LIN {X 0,Y 409.441,Z 300.015,A -85,B 0,C 180,E1 20196.049,E2 20196.049} C_VEL
LIN {X 0,Y 414.724,Z 318.91,A -85,B 0,C 180,E1 20192.601,E2 20192.601} C_VEL
LIN {X 0,Y 418.391,Z 333.673,A -85,B 0,C 180,E1 20190.048,E2 20190.048} C_VEL
LIN {X 0,Y 416.064,Z 361.542,A -85,B 0,C 180,E1 20186.001,E2 20186.001} C_VEL
LIN {X 0,Y 414.003,Z 389.743,A -85,B 0,C 180,E1 20181.965,E2 20181.965} C_VEL
LIN {X 0,Y 413.216,Z 403.009,A -85,B 0,C 180,E1 20180.124,E2 20180.124} C_VEL
LIN {X 0,Y 416.515,Z 427.421,A -85,B 0,C 180,E1 20179.379,E2 20179.379} C_VEL
LIN {X 0,Y 413.998,Z 526.951,A -85,B 0,C 180,E1 20177.125,E2 20177.125} C_VEL
LIN {X 0,Y 413.552,Z 542.343,A -85,B 0,C 180,E1 20176.538,E2 20176.538} C_VEL
LIN {X 0,Y 412.934,Z 558.221,A -85,B 0,C 180,E1 20175.661,E2 20175.661} C_VEL
LIN {X 0,Y 412.172,Z 574.05,A -85,B 0,C 180,E1 20174.467,E2 20174.467} C_VEL
LIN {X 0,Y 411.427,Z 588.228,A -85,B 0,C 180,E1 20173.06,E2 20173.06} C_VEL
LIN {X 0,Y 410.741,Z 600.404,A -85,B 0,C 180,E1 20171.512,E2 20171.512} C_VEL
LIN {X 0,Y 410.206,Z 610.147,A -85,B 0,C 180,E1 20169.963,E2 20169.963} C_VEL
LIN {X 0,Y 409.748,Z 619.266,A -85,B 0,C 180,E1 20168.134,E2 20168.134} C_VEL
LIN {X 0,Y 409.435,Z 626.69,A -85,B 0,C 180,E1 20166.166,E2 20166.166} C_VEL
LIN {X 0,Y 409.281,Z 631.788,A -85,B 0,C 180,E1 20164.341,E2 20164.341} C_VEL
LIN {X 0,Y 409.227,Z 635.7,A -85,B 0,C 180,E1 20162.238,E2 20162.238} C_VEL
LIN {X 0,Y 409.285,Z 637.574,A -85,B 0,C 180,E1 20160.278,E2 20160.278} C_VEL
LIN {X 0,Y 409.451,Z 637.785,A -85,B 0,C 180,E1 20158.179,E2 20158.179} C_VEL
LIN {X 0,Y 409.729,Z 636.027,A -85,B 0,C 180,E1 20156.08,E2 20156.08} C_VEL
LIN {X 0,Y 410.14,Z 632.531,A -85,B 0,C 180,E1 20154.073,E2 20154.073} C_VEL
LIN {X 0,Y 410.724,Z 626.914,A -85,B 0,C 180,E1 20152.022,E2 20152.022} C_VEL
LIN {X 0,Y 411.417,Z 619.96,A -85,B 0,C 180,E1 20150.203,E2 20150.203} C_VEL
LIN {X 0,Y 412.286,Z 611.32,A -85,B 0,C 180,E1 20148.457,E2 20148.457} C_VEL
LIN {X 0,Y 413.331,Z 600.124,A -85,B 0,C 180,E1 20146.713,E2 20146.713} C_VEL
LIN {X 0,Y 414.344,Z 588.102,A -85,B 0,C 180,E1 20145.249,E2 20145.249} C_VEL
LIN {X 0,Y 415.388,Z 575.258,A -85,B 0,C 180,E1 20144,E2 20144} C_VEL
LIN {X 0,Y 416.433,Z 560.28,A -85,B 0,C 180,E1 20142.865,E2 20142.865} C_VEL
LIN {X 0,Y 417.393,Z 543.508,A -85,B 0,C 180,E1 20141.926,E2 20141.926} C_VEL
LIN {X 0,Y 418.191,Z 525.443,A -85,B 0,C 180,E1 20141.231,E2 20141.231} C_VEL
LIN {X 0,Y 424.218,Z 435.023,A -85,B 0,C 180,E1 20138.466,E2 20138.466} C_VEL
LIN {X 0,Y 424.373,Z 429.953,A -85,B 0,C 180,E1 20138.28,E2 20138.28} C_VEL
LIN {X 0,Y 421.463,Z 411.862,A -85,B 0,C 180,E1 20137.24,E2 20137.24} C_VEL
LIN {X 0,Y 419.727,Z 402.661,A -85,B 0,C 180,E1 20136.631,E2 20136.631} C_VEL
LIN {X 0,Y 423.555,Z 377.639,A -85,B 0,C 180,E1 20132.575,E2 20132.575} C_VEL
LIN {X 0,Y 428.286,Z 354.651,A -85,B 0,C 180,E1 20128.626,E2 20128.626} C_VEL
LIN {X 0,Y 429.025,Z 351.42,A -85,B 0,C 180,E1 20128.03,E2 20128.03} C_VEL
LIN {X 0,Y 427.636,Z 343.386,A -85,B 0,C 180,E1 20125.701,E2 20125.701} C_VEL
LIN {X 0,Y 426.273,Z 337.13,A -85,B 0,C 180,E1 20123.341,E2 20123.341} C_VEL
LIN {X 0,Y 425.312,Z 333.711,A -85,B 0,C 180,E1 20121.523,E2 20121.523} C_VEL
LIN {X 0,Y 424.901,Z 331.733,A -85,B 0,C 180,E1 20120.098,E2 20120.098} C_VEL
LIN {X 0,Y 424.618,Z 330.119,A -85,B 0,C 180,E1 20117.48,E2 20117.48} C_VEL
LIN {X 0,Y 424.896,Z 330.575,A -85,B 0,C 180,E1 20115.66,E2 20115.66} C_VEL
LIN {X 0,Y 426.204,Z 333.163,A -85,B 0,C 180,E1 20113.146,E2 20113.146} C_VEL
LIN {X 0,Y 427.711,Z 337.595,A -85,B 0,C 180,E1 20111.064,E2 20111.064} C_VEL
LIN {X 0,Y 429.535,Z 343.22,A -85,B 0,C 180,E1 20109.18,E2 20109.18} C_VEL
LIN {X 0,Y 431.487,Z 350.329,A -85,B 0,C 180,E1 20107.361,E2 20107.361} C_VEL
LIN {X 0,Y 432.028,Z 352.863,A -85,B 0,C 180,E1 20106.829,E2 20106.829} C_VEL
LIN {X 0,Y 426.646,Z 376.903,A -85,B 0,C 180,E1 20103.902,E2 20103.902} C_VEL
LIN {X 0,Y 424.049,Z 392.881,A -85,B 0,C 180,E1 20102.112,E2 20102.112} C_VEL
LIN {X 0,Y 425.783,Z 409.021,A -85,B 0,C 180,E1 20101.466,E2 20101.466} C_VEL
LIN {X 0,Y 425.816,Z 416.278,A -85,B 0,C 180,E1 20101.257,E2 20101.257} C_VEL
LIN {X 0,Y 421.996,Z 515.171,A -85,B 0,C 180,E1 20099.047,E2 20099.047} C_VEL
LIN {X 0,Y 419.948,Z 585.828,A -85,B 0,C 180,E1 20097.578,E2 20097.578} C_VEL
LIN {X 0,Y 418.736,Z 605.858,A -85,B 0,C 180,E1 20096.904,E2 20096.904} C_VEL
LIN {X 0,Y 417.429,Z 623.258,A -85,B 0,C 180,E1 20096.072,E2 20096.072} C_VEL
LIN {X 0,Y 415.921,Z 641.014,A -85,B 0,C 180,E1 20094.963,E2 20094.963} C_VEL
LIN {X 0,Y 414.353,Z 658.072,A -85,B 0,C 180,E1 20093.615,E2 20093.615} C_VEL
LIN {X 0,Y 412.829,Z 674.111,A -85,B 0,C 180,E1 20092.05,E2 20092.05} C_VEL
LIN {X 0,Y 411.475,Z 689.013,A -85,B 0,C 180,E1 20090.287,E2 20090.287} C_VEL
LIN {X 0,Y 410.322,Z 702.807,A -85,B 0,C 180,E1 20088.322,E2 20088.322} C_VEL
LIN {X 0,Y 409.422,Z 715.375,A -85,B 0,C 180,E1 20086.166,E2 20086.166} C_VEL
LIN {X 0,Y 408.847,Z 726.454,A -85,B 0,C 180,E1 20083.856,E2 20083.856} C_VEL
LIN {X 0,Y 408.556,Z 735.338,A -85,B 0,C 180,E1 20081.578,E2 20081.578} C_VEL
LIN {X 0,Y 408.504,Z 742.848,A -85,B 0,C 180,E1 20079.155,E2 20079.155} C_VEL
LIN {X 0,Y 408.585,Z 748.491,A -85,B 0,C 180,E1 20076.747,E2 20076.747} C_VEL
LIN {X 0,Y 408.725,Z 752.398,A -85,B 0,C 180,E1 20074.35,E2 20074.35} C_VEL
LIN {X 0,Y 408.841,Z 754.641,A -85,B 0,C 180,E1 20071.963,E2 20071.963} C_VEL
LIN {X 0,Y 408.862,Z 755.26,A -85,B 0,C 180,E1 20069.581,E2 20069.581} C_VEL
LIN {X 0,Y 408.779,Z 754.252,A -85,B 0,C 180,E1 20067.197,E2 20067.197} C_VEL
LIN {X 0,Y 408.628,Z 751.594,A -85,B 0,C 180,E1 20064.801,E2 20064.801} C_VEL
LIN {X 0,Y 408.496,Z 747.256,A -85,B 0,C 180,E1 20062.406,E2 20062.406} C_VEL
LIN {X 0,Y 408.465,Z 741.108,A -85,B 0,C 180,E1 20059.992,E2 20059.992} C_VEL
LIN {X 0,Y 408.614,Z 732.997,A -85,B 0,C 180,E1 20057.566,E2 20057.566} C_VEL
LIN {X 0,Y 409.04,Z 723.353,A -85,B 0,C 180,E1 20055.274,E2 20055.274} C_VEL
LIN {X 0,Y 409.742,Z 711.86,A -85,B 0,C 180,E1 20053.054,E2 20053.054} C_VEL
LIN {X 0,Y 410.71,Z 699.143,A -85,B 0,C 180,E1 20051.036,E2 20051.036} C_VEL
LIN {X 0,Y 411.906,Z 684.831,A -85,B 0,C 180,E1 20049.157,E2 20049.157} C_VEL
LIN {X 0,Y 413.227,Z 669.717,A -85,B 0,C 180,E1 20047.525,E2 20047.525} C_VEL
LIN {X 0,Y 414.612,Z 653.545,A -85,B 0,C 180,E1 20046.101,E2 20046.101} C_VEL
LIN {X 0,Y 415.964,Z 636.517,A -85,B 0,C 180,E1 20044.898,E2 20044.898} C_VEL
LIN {X 0,Y 417.227,Z 618.592,A -85,B 0,C 180,E1 20043.914,E2 20043.914} C_VEL
LIN {X 0,Y 418.356,Z 599.425,A -85,B 0,C 180,E1 20043.148,E2 20043.148} C_VEL
LIN {X 0,Y 419.065,Z 580.405,A -85,B 0,C 180,E1 20042.65,E2 20042.65} C_VEL
LIN {X 0,Y 422.694,Z 411.284,A -85,B 0,C 180,E1 20039.443,E2 20039.443} C_VEL
LIN {X 0,Y 420.158,Z 388.361,A -85,B 0,C 180,E1 20038.811,E2 20038.811} C_VEL
LIN {X 0,Y 424.415,Z 345.859,A -85,B 0,C 180,E1 20034.601,E2 20034.601} C_VEL
LIN {X 0,Y 424.551,Z 343.397,A -85,B 0,C 180,E1 20034.343,E2 20034.343} C_VEL
LIN {X 0,Y 416.406,Z 319.629,A -85,B 0,C 180,E1 20031.017,E2 20031.017} C_VEL
LIN {X 0,Y 409.402,Z 299.802,A -85,B 0,C 180,E1 20027.998,E2 20027.998} C_VEL
LIN {X 0,Y 409.391,Z 299.803,A -85,B 0,C 180,E1 20024.109,E2 20024.109} C_VEL
LIN {X 0,Y 409.376,Z 299.804,A -85,B 0,C 180,E1 20020.335,E2 20020.335} C_VEL
LIN {X 0,Y 409.367,Z 299.801,A -85,B 0,C 180,E1 20016.53,E2 20016.53} C_VEL
LIN {X 0,Y 409.368,Z 299.8,A -85,B 0,C 180,E1 20012.67,E2 20012.67} C_VEL
LIN {X 0,Y 409.371,Z 299.8,A -85,B 0,C 180,E1 20008.74,E2 20008.74} C_VEL
LIN {X 0,Y 409.373,Z 299.8,A -85,B 0,C 180,E1 20004.842,E2 20004.842} C_VEL
LIN {X 0,Y 409.381,Z 299.8,A -85,B 0,C 180,E1 20001.042,E2 20001.042} C_VEL
LIN {X 0,Y 409.398,Z 299.799,A -85,B 0,C 180,E1 19997.273,E2 19997.273} C_VEL
LIN {X 0,Y 409.423,Z 299.8,A -85,B 0,C 180,E1 19993.561,E2 19993.561} C_VEL
LIN {X 0,Y 409.42,Z 299.8,A -85,B 0,C 180,E1 19989.561,E2 19989.561} C_VEL
LIN {X 0,Y 409.416,Z 299.801,A -85,B 0,C 180,E1 19985.748,E2 19985.748} C_VEL
LIN {X 0,Y 409.411,Z 299.8,A -85,B 0,C 180,E1 19981.821,E2 19981.821} C_VEL
LIN {X 0,Y 409.393,Z 299.8,A -85,B 0,C 180,E1 19978.043,E2 19978.043} C_VEL
LIN {X 0,Y 409.382,Z 299.8,A -85,B 0,C 180,E1 19974.255,E2 19974.255} C_VEL
LIN {X 0,Y 409.379,Z 299.799,A -85,B 0,C 180,E1 19970.442,E2 19970.442} C_VEL
LIN {X 0,Y 409.381,Z 299.799,A -85,B 0,C 180,E1 19966.586,E2 19966.586} C_VEL
LIN {X 0,Y 409.386,Z 299.798,A -85,B 0,C 180,E1 19962.733,E2 19962.733} C_VEL
LIN {X 0,Y 409.393,Z 299.798,A -85,B 0,C 180,E1 19958.897,E2 19958.897} C_VEL
LIN {X 0,Y 409.414,Z 299.797,A -85,B 0,C 180,E1 19955.165,E2 19955.165} C_VEL
LIN {X 0,Y 409.424,Z 299.797,A -85,B 0,C 180,E1 19951.246,E2 19951.246} C_VEL
LIN {X 0,Y 409.431,Z 299.798,A -85,B 0,C 180,E1 19947.34,E2 19947.34} C_VEL
LIN {X 0,Y 409.43,Z 299.799,A -85,B 0,C 180,E1 19943.429,E2 19943.429} C_VEL
LIN {X 0,Y 409.437,Z 299.799,A -85,B 0,C 180,E1 19939.494,E2 19939.494} C_VEL
LIN {X 0,Y 409.428,Z 299.8,A -85,B 0,C 180,E1 19935.485,E2 19935.485} C_VEL
LIN {X 0,Y 409.423,Z 299.8,A -85,B 0,C 180,E1 19931.624,E2 19931.624} C_VEL
LIN {X 0,Y 409.401,Z 299.799,A -85,B 0,C 180,E1 19927.927,E2 19927.927} C_VEL
LIN {X 0,Y 409.395,Z 299.798,A -85,B 0,C 180,E1 19924.118,E2 19924.118} C_VEL
LIN {X 0,Y 409.394,Z 299.798,A -85,B 0,C 180,E1 19920.205,E2 19920.205} C_VEL
LIN {X 0,Y 409.394,Z 299.797,A -85,B 0,C 180,E1 19916.329,E2 19916.329} C_VEL
LIN {X 0,Y 409.395,Z 299.797,A -85,B 0,C 180,E1 19912.394,E2 19912.394} C_VEL
LIN {X 0,Y 409.398,Z 299.797,A -85,B 0,C 180,E1 19908.51,E2 19908.51} C_VEL
LIN {X 0,Y 409.406,Z 299.796,A -85,B 0,C 180,E1 19904.713,E2 19904.713} C_VEL
LIN {X 0,Y 409.426,Z 299.796,A -85,B 0,C 180,E1 19900.98,E2 19900.98} C_VEL
LIN {X 0,Y 409.445,Z 299.795,A -85,B 0,C 180,E1 19897.153,E2 19897.153} C_VEL
LIN {X 0,Y 409.436,Z 299.797,A -85,B 0,C 180,E1 19893.219,E2 19893.219} C_VEL
LIN {X 0,Y 409.445,Z 299.797,A -85,B 0,C 180,E1 19889.299,E2 19889.299} C_VEL
LIN {X 0,Y 409.432,Z 299.8,A -85,B 0,C 180,E1 19885.377,E2 19885.377} C_VEL
LIN {X 0,Y 409.428,Z 299.799,A -85,B 0,C 180,E1 19881.489,E2 19881.489} C_VEL
LIN {X 0,Y 409.412,Z 299.798,A -85,B 0,C 180,E1 19877.741,E2 19877.741} C_VEL
LIN {X 0,Y 408.478,Z 299.923,A -85,B 0,C 180,E1 19876.663,E2 19876.663} C_VEL
LIN {X 0,Y 403.736,Z 300.514,A -85,B 0,C 180,E1 19874.553,E2 19874.553} C_VEL
LIN {X 0,Y 401.598,Z 300.773,A -85,B 0,C 180,E1 19873.149,E2 19873.149} C_VEL
LIN {X 0,Y 401.49,Z 300.784,A -85,B 0,C 180,E1 19872.83,E2 19872.83} C_VEL
LIN {X 0,Y 401.505,Z 300.783,A -85,B 0,C 180,E1 19868.985,E2 19868.985} C_VEL
LIN {X 0,Y 401.503,Z 300.784,A -85,B 0,C 180,E1 19865.014,E2 19865.014} C_VEL
LIN {X 0,Y 401.511,Z 300.784,A -85,B 0,C 180,E1 19861.11,E2 19861.11} C_VEL
LIN {X 0,Y 401.505,Z 300.785,A -85,B 0,C 180,E1 19857.119,E2 19857.119} C_VEL
LIN {X 0,Y 401.505,Z 300.784,A -85,B 0,C 180,E1 19853.066,E2 19853.066} C_VEL
LIN {X 0,Y 401.509,Z 300.784,A -85,B 0,C 180,E1 19849.084,E2 19849.084} C_VEL
LIN {X 0,Y 401.5,Z 300.788,A -85,B 0,C 180,E1 19845.189,E2 19845.189} C_VEL
LIN {X 0,Y 401.505,Z 300.787,A -85,B 0,C 180,E1 19841.229,E2 19841.229} C_VEL
LIN {X 0,Y 401.491,Z 300.788,A -85,B 0,C 180,E1 19837.397,E2 19837.397} C_VEL
LIN {X 0,Y 401.503,Z 300.865,A -85,B 0,C 180,E1 19836.611,E2 19836.611} C_VEL
LIN {X 0,Y 406.949,Z 320.456,A -85,B 0,C 180,E1 19832.968,E2 19832.968} C_VEL
LIN {X 0,Y 410.79,Z 335.895,A -85,B 0,C 180,E1 19830.251,E2 19830.251} C_VEL
LIN {X 0,Y 408.357,Z 363.768,A -85,B 0,C 180,E1 19826.147,E2 19826.147} C_VEL
LIN {X 0,Y 406.149,Z 392.506,A -85,B 0,C 180,E1 19821.972,E2 19821.972} C_VEL
LIN {X 0,Y 405.523,Z 402.833,A -85,B 0,C 180,E1 19820.519,E2 19820.519} C_VEL
LIN {X 0,Y 408.911,Z 428.375,A -85,B 0,C 180,E1 19819.715,E2 19819.715} C_VEL
LIN {X 0,Y 406.252,Z 527.745,A -85,B 0,C 180,E1 19817.392,E2 19817.392} C_VEL
LIN {X 0,Y 405.756,Z 543.832,A -85,B 0,C 180,E1 19816.754,E2 19816.754} C_VEL
LIN {X 0,Y 405.144,Z 558.966,A -85,B 0,C 180,E1 19815.896,E2 19815.896} C_VEL
LIN {X 0,Y 404.354,Z 574.826,A -85,B 0,C 180,E1 19814.68,E2 19814.68} C_VEL
LIN {X 0,Y 403.579,Z 589.06,A -85,B 0,C 180,E1 19813.246,E2 19813.246} C_VEL
LIN {X 0,Y 402.841,Z 601.812,A -85,B 0,C 180,E1 19811.596,E2 19811.596} C_VEL
LIN {X 0,Y 402.245,Z 612.27,A -85,B 0,C 180,E1 19809.873,E2 19809.873} C_VEL
LIN {X 0,Y 401.822,Z 620.594,A -85,B 0,C 180,E1 19808.152,E2 19808.152} C_VEL
LIN {X 0,Y 401.507,Z 628.02,A -85,B 0,C 180,E1 19806.145,E2 19806.145} C_VEL
LIN {X 0,Y 401.345,Z 633.398,A -85,B 0,C 180,E1 19804.141,E2 19804.141} C_VEL
LIN {X 0,Y 401.31,Z 636.994,A -85,B 0,C 180,E1 19802.14,E2 19802.14} C_VEL
LIN {X 0,Y 401.387,Z 638.913,A -85,B 0,C 180,E1 19799.998,E2 19799.998} C_VEL
LIN {X 0,Y 401.58,Z 639.044,A -85,B 0,C 180,E1 19798,E2 19798} C_VEL
LIN {X 0,Y 401.9,Z 637.26,A -85,B 0,C 180,E1 19795.861,E2 19795.861} C_VEL
LIN {X 0,Y 402.347,Z 633.821,A -85,B 0,C 180,E1 19793.864,E2 19793.864} C_VEL
LIN {X 0,Y 402.968,Z 628.538,A -85,B 0,C 180,E1 19791.868,E2 19791.868} C_VEL
LIN {X 0,Y 403.732,Z 621.742,A -85,B 0,C 180,E1 19790.015,E2 19790.015} C_VEL
LIN {X 0,Y 404.704,Z 612.815,A -85,B 0,C 180,E1 19788.165,E2 19788.165} C_VEL
LIN {X 0,Y 405.895,Z 601.238,A -85,B 0,C 180,E1 19786.319,E2 19786.319} C_VEL
LIN {X 0,Y 407.068,Z 588.654,A -85,B 0,C 180,E1 19784.761,E2 19784.761} C_VEL
LIN {X 0,Y 408.191,Z 575.598,A -85,B 0,C 180,E1 19783.491,E2 19783.491} C_VEL
LIN {X 0,Y 409.297,Z 560.926,A -85,B 0,C 180,E1 19782.366,E2 19782.366} C_VEL
LIN {X 0,Y 410.316,Z 545.116,A -85,B 0,C 180,E1 19781.449,E2 19781.449} C_VEL
LIN {X 0,Y 411.2,Z 527.167,A -85,B 0,C 180,E1 19780.724,E2 19780.724} C_VEL
LIN {X 0,Y 418.014,Z 433.46,A -85,B 0,C 180,E1 19777.747,E2 19777.747} C_VEL
LIN {X 0,Y 416.157,Z 419.167,A -85,B 0,C 180,E1 19776.928,E2 19776.928} C_VEL
LIN {X 0,Y 413.134,Z 402.466,A -85,B 0,C 180,E1 19775.78,E2 19775.78} C_VEL
LIN {X 0,Y 417.403,Z 377.958,A -85,B 0,C 180,E1 19771.685,E2 19771.685} C_VEL
LIN {X 0,Y 422.437,Z 356.26,A -85,B 0,C 180,E1 19767.821,E2 19767.821} C_VEL
LIN {X 0,Y 422.44,Z 354.305,A -85,B 0,C 180,E1 19767.339,E2 19767.339} C_VEL
LIN {X 0,Y 421.315,Z 347.222,A -85,B 0,C 180,E1 19765.113,E2 19765.113} C_VEL
LIN {X 0,Y 420.202,Z 341.819,A -85,B 0,C 180,E1 19762.857,E2 19762.857} C_VEL
LIN {X 0,Y 419.509,Z 338.644,A -85,B 0,C 180,E1 19760.987,E2 19760.987} C_VEL
LIN {X 0,Y 419.266,Z 337.346,A -85,B 0,C 180,E1 19759.916,E2 19759.916} C_VEL
LIN {X 0,Y 419.215,Z 335.944,A -85,B 0,C 180,E1 19757.175,E2 19757.175} C_VEL
LIN {X 0,Y 419.561,Z 336.796,A -85,B 0,C 180,E1 19755.25,E2 19755.25} C_VEL
LIN {X 0,Y 420.818,Z 339.472,A -85,B 0,C 180,E1 19752.961,E2 19752.961} C_VEL
LIN {X 0,Y 422.108,Z 343.366,A -85,B 0,C 180,E1 19751.125,E2 19751.125} C_VEL
LIN {X 0,Y 424.055,Z 349.661,A -85,B 0,C 180,E1 19749.018,E2 19749.018} C_VEL
LIN {X 0,Y 425.699,Z 356.545,A -85,B 0,C 180,E1 19747.3,E2 19747.3} C_VEL
LIN {X 0,Y 419.973,Z 380.043,A -85,B 0,C 180,E1 19744.351,E2 19744.351} C_VEL
LIN {X 0,Y 417.641,Z 393.224,A -85,B 0,C 180,E1 19742.833,E2 19742.833} C_VEL
LIN {X 0,Y 419.323,Z 408.99,A -85,B 0,C 180,E1 19742.147,E2 19742.147} C_VEL
LIN {X 0,Y 419.446,Z 416.244,A -85,B 0,C 180,E1 19741.917,E2 19741.917} C_VEL
LIN {X 0,Y 415.269,Z 512.08,A -85,B 0,C 180,E1 19739.687,E2 19739.687} C_VEL
LIN {X 0,Y 412.858,Z 585.335,A -85,B 0,C 180,E1 19738.098,E2 19738.098} C_VEL
LIN {X 0,Y 411.556,Z 605.144,A -85,B 0,C 180,E1 19737.411,E2 19737.411} C_VEL
LIN {X 0,Y 410.073,Z 623.422,A -85,B 0,C 180,E1 19736.511,E2 19736.511} C_VEL
LIN {X 0,Y 408.439,Z 641.077,A -85,B 0,C 180,E1 19735.367,E2 19735.367} C_VEL
LIN {X 0,Y 406.694,Z 658.491,A -85,B 0,C 180,E1 19733.933,E2 19733.933} C_VEL
LIN {X 0,Y 405.084,Z 674.231,A -85,B 0,C 180,E1 19732.342,E2 19732.342} C_VEL
LIN {X 0,Y 403.544,Z 690.013,A -85,B 0,C 180,E1 19730.397,E2 19730.397} C_VEL
LIN {X 0,Y 402.352,Z 703.428,A -85,B 0,C 180,E1 19728.398,E2 19728.398} C_VEL
LIN {X 0,Y 401.428,Z 715.696,A -85,B 0,C 180,E1 19726.199,E2 19726.199} C_VEL
LIN {X 0,Y 400.845,Z 726.469,A -85,B 0,C 180,E1 19723.856,E2 19723.856} C_VEL
LIN {X 0,Y 400.55,Z 735.646,A -85,B 0,C 180,E1 19721.374,E2 19721.374} C_VEL
LIN {X 0,Y 400.534,Z 742.819,A -85,B 0,C 180,E1 19718.905,E2 19718.905} C_VEL
LIN {X 0,Y 400.642,Z 748.165,A -85,B 0,C 180,E1 19716.449,E2 19716.449} C_VEL
LIN {X 0,Y 400.807,Z 751.795,A -85,B 0,C 180,E1 19714.006,E2 19714.006} C_VEL
LIN {X 0,Y 400.926,Z 753.752,A -85,B 0,C 180,E1 19711.573,E2 19711.573} C_VEL
LIN {X 0,Y 400.944,Z 754.057,A -85,B 0,C 180,E1 19709.144,E2 19709.144} C_VEL
LIN {X 0,Y 400.827,Z 752.717,A -85,B 0,C 180,E1 19706.712,E2 19706.712} C_VEL
LIN {X 0,Y 400.663,Z 749.719,A -85,B 0,C 180,E1 19704.272,E2 19704.272} C_VEL
LIN {X 0,Y 400.525,Z 744.996,A -85,B 0,C 180,E1 19701.821,E2 19701.821} C_VEL
LIN {X 0,Y 400.507,Z 738.437,A -85,B 0,C 180,E1 19699.355,E2 19699.355} C_VEL
LIN {X 0,Y 400.707,Z 730.421,A -85,B 0,C 180,E1 19697.024,E2 19697.024} C_VEL
LIN {X 0,Y 401.187,Z 720.393,A -85,B 0,C 180,E1 19694.683,E2 19694.683} C_VEL
LIN {X 0,Y 401.965,Z 708.826,A -85,B 0,C 180,E1 19692.485,E2 19692.485} C_VEL
LIN {X 0,Y 403.035,Z 695.667,A -85,B 0,C 180,E1 19690.434,E2 19690.434} C_VEL
LIN {X 0,Y 404.277,Z 681.457,A -85,B 0,C 180,E1 19688.606,E2 19688.606} C_VEL
LIN {X 0,Y 405.711,Z 665.612,A -85,B 0,C 180,E1 19686.932,E2 19686.932} C_VEL
LIN {X 0,Y 407.2,Z 648.692,A -85,B 0,C 180,E1 19685.484,E2 19685.484} C_VEL
LIN {X 0,Y 408.576,Z 631.813,A -85,B 0,C 180,E1 19684.334,E2 19684.334} C_VEL
LIN {X 0,Y 409.867,Z 613.454,A -85,B 0,C 180,E1 19683.37,E2 19683.37} C_VEL
LIN {X 0,Y 410.95,Z 594.557,A -85,B 0,C 180,E1 19682.663,E2 19682.663} C_VEL
LIN {X 0,Y 411.592,Z 574.104,A -85,B 0,C 180,E1 19682.184,E2 19682.184} C_VEL
LIN {X 0,Y 415.286,Z 412.136,A -85,B 0,C 180,E1 19679.039,E2 19679.039} C_VEL
LIN {X 0,Y 412.724,Z 388.405,A -85,B 0,C 180,E1 19678.368,E2 19678.368} C_VEL
LIN {X 0,Y 417.22,Z 346.226,A -85,B 0,C 180,E1 19674.098,E2 19674.098} C_VEL
LIN {X 0,Y 409.155,Z 322.58,A -85,B 0,C 180,E1 19670.736,E2 19670.736} C_VEL
LIN {X 0,Y 401.448,Z 300.792,A -85,B 0,C 180,E1 19667.357,E2 19667.357} C_VEL
LIN {X 0,Y 401.456,Z 300.791,A -85,B 0,C 180,E1 19663.426,E2 19663.426} C_VEL
LIN {X 0,Y 401.474,Z 300.791,A -85,B 0,C 180,E1 19659.612,E2 19659.612} C_VEL
LIN {X 0,Y 401.473,Z 300.79,A -85,B 0,C 180,E1 19655.647,E2 19655.647} C_VEL
LIN {X 0,Y 401.476,Z 300.79,A -85,B 0,C 180,E1 19651.601,E2 19651.601} C_VEL
LIN {X 0,Y 401.478,Z 300.79,A -85,B 0,C 180,E1 19647.758,E2 19647.758} C_VEL
LIN {X 0,Y 401.476,Z 300.79,A -85,B 0,C 180,E1 19643.796,E2 19643.796} C_VEL
LIN {X 0,Y 401.463,Z 300.789,A -85,B 0,C 180,E1 19639.952,E2 19639.952} C_VEL
LIN {X 0,Y 401.455,Z 300.789,A -85,B 0,C 180,E1 19636.05,E2 19636.05} C_VEL
LIN {X 0,Y 401.444,Z 300.789,A -85,B 0,C 180,E1 19632.224,E2 19632.224} C_VEL
LIN {X 0,Y 401.436,Z 300.789,A -85,B 0,C 180,E1 19628.452,E2 19628.452} C_VEL
LIN {X 0,Y 401.437,Z 300.789,A -85,B 0,C 180,E1 19624.573,E2 19624.573} C_VEL
LIN {X 0,Y 401.437,Z 300.788,A -85,B 0,C 180,E1 19620.573,E2 19620.573} C_VEL
LIN {X 0,Y 401.439,Z 300.788,A -85,B 0,C 180,E1 19616.575,E2 19616.575} C_VEL
LIN {X 0,Y 401.44,Z 300.788,A -85,B 0,C 180,E1 19612.561,E2 19612.561} C_VEL
LIN {X 0,Y 401.441,Z 300.788,A -85,B 0,C 180,E1 19608.655,E2 19608.655} C_VEL
LIN {X 0,Y 401.449,Z 300.787,A -85,B 0,C 180,E1 19604.842,E2 19604.842} C_VEL
LIN {X 0,Y 401.457,Z 300.787,A -85,B 0,C 180,E1 19600.96,E2 19600.96} C_VEL
LIN {X 0,Y 401.472,Z 300.787,A -85,B 0,C 180,E1 19597.14,E2 19597.14} C_VEL
LIN {X 0,Y 401.479,Z 300.786,A -85,B 0,C 180,E1 19593.21,E2 19593.21} C_VEL
LIN {X 0,Y 401.491,Z 300.786,A -85,B 0,C 180,E1 19589.304,E2 19589.304} C_VEL
LIN {X 0,Y 401.489,Z 300.788,A -85,B 0,C 180,E1 19585.406,E2 19585.406} C_VEL
LIN {X 0,Y 401.5,Z 300.787,A -85,B 0,C 180,E1 19581.438,E2 19581.438} C_VEL
LIN {X 0,Y 401.491,Z 300.789,A -85,B 0,C 180,E1 19577.487,E2 19577.487} C_VEL
LIN {X 0,Y 401.485,Z 300.789,A -85,B 0,C 180,E1 19573.56,E2 19573.56} C_VEL
LIN {X 0,Y 401.487,Z 300.788,A -85,B 0,C 180,E1 19569.607,E2 19569.607} C_VEL
LIN {X 0,Y 401.479,Z 300.789,A -85,B 0,C 180,E1 19565.643,E2 19565.643} C_VEL
LIN {X 0,Y 401.467,Z 300.788,A -85,B 0,C 180,E1 19561.868,E2 19561.868} C_VEL
LIN {X 0,Y 401.459,Z 300.787,A -85,B 0,C 180,E1 19558.079,E2 19558.079} C_VEL
LIN {X 0,Y 401.456,Z 300.786,A -85,B 0,C 180,E1 19554.263,E2 19554.263} C_VEL
LIN {X 0,Y 401.457,Z 300.786,A -85,B 0,C 180,E1 19550.253,E2 19550.253} C_VEL
LIN {X 0,Y 401.456,Z 300.786,A -85,B 0,C 180,E1 19546.345,E2 19546.345} C_VEL
LIN {X 0,Y 401.46,Z 300.786,A -85,B 0,C 180,E1 19542.513,E2 19542.513} C_VEL
LIN {X 0,Y 401.464,Z 300.785,A -85,B 0,C 180,E1 19538.593,E2 19538.593} C_VEL
LIN {X 0,Y 401.48,Z 300.785,A -85,B 0,C 180,E1 19534.856,E2 19534.856} C_VEL
LIN {X 0,Y 401.497,Z 300.784,A -85,B 0,C 180,E1 19530.998,E2 19530.998} C_VEL
LIN {X 0,Y 401.498,Z 300.785,A -85,B 0,C 180,E1 19527.144,E2 19527.144} C_VEL
LIN {X 0,Y 401.51,Z 300.784,A -85,B 0,C 180,E1 19523.134,E2 19523.134} C_VEL
LIN {X 0,Y 401.499,Z 300.785,A -85,B 0,C 180,E1 19519.089,E2 19519.089} C_VEL
LIN {X 0,Y 401.507,Z 300.783,A -85,B 0,C 180,E1 19515.053,E2 19515.053} C_VEL
LIN {X 0,Y 401.49,Z 300.784,A -85,B 0,C 180,E1 19512.83,E2 19512.83} C_VEL
LIN {X 0,Y 400.457,Z 300.915,A -85,B 0,C 180,E1 19511.731,E2 19511.731} C_VEL
LIN {X 0,Y 393.94,Z 301.725,A -85,B 0,C 180,E1 19508.551,E2 19508.551} C_VEL
LIN {X 0,Y 393.531,Z 301.775,A -85,B 0,C 180,E1 19507.822,E2 19507.822} C_VEL
LIN {X 0,Y 393.531,Z 301.775,A -85,B 0,C 180,E1 19503.924,E2 19503.924} C_VEL
LIN {X 0,Y 393.53,Z 301.775,A -85,B 0,C 180,E1 19499.964,E2 19499.964} C_VEL
LIN {X 0,Y 393.528,Z 301.774,A -85,B 0,C 180,E1 19496.015,E2 19496.015} C_VEL
LIN {X 0,Y 393.53,Z 301.774,A -85,B 0,C 180,E1 19491.959,E2 19491.959} C_VEL
LIN {X 0,Y 393.532,Z 301.774,A -85,B 0,C 180,E1 19488.07,E2 19488.07} C_VEL
LIN {X 0,Y 393.533,Z 301.775,A -85,B 0,C 180,E1 19484.025,E2 19484.025} C_VEL
LIN {X 0,Y 393.533,Z 301.778,A -85,B 0,C 180,E1 19479.997,E2 19479.997} C_VEL
LIN {X 0,Y 393.585,Z 301.947,A -85,B 0,C 180,E1 19477.151,E2 19477.151} C_VEL
LIN {X 0,Y 399.047,Z 321.425,A -85,B 0,C 180,E1 19473.448,E2 19473.448} C_VEL
LIN {X 0,Y 403.212,Z 337.52,A -85,B 0,C 180,E1 19470.551,E2 19470.551} C_VEL
LIN {X 0,Y 400.775,Z 364.464,A -85,B 0,C 180,E1 19466.521,E2 19466.521} C_VEL
LIN {X 0,Y 398.482,Z 392.78,A -85,B 0,C 180,E1 19462.34,E2 19462.34} C_VEL
LIN {X 0,Y 397.843,Z 402.762,A -85,B 0,C 180,E1 19460.918,E2 19460.918} C_VEL
LIN {X 0,Y 401.313,Z 429.19,A -85,B 0,C 180,E1 19460.062,E2 19460.062} C_VEL
LIN {X 0,Y 398.518,Z 528.363,A -85,B 0,C 180,E1 19457.675,E2 19457.675} C_VEL
LIN {X 0,Y 398.026,Z 543.876,A -85,B 0,C 180,E1 19457.052,E2 19457.052} C_VEL
LIN {X 0,Y 397.361,Z 559.711,A -85,B 0,C 180,E1 19456.141,E2 19456.141} C_VEL
LIN {X 0,Y 396.54,Z 575.601,A -85,B 0,C 180,E1 19454.901,E2 19454.901} C_VEL
LIN {X 0,Y 395.736,Z 589.891,A -85,B 0,C 180,E1 19453.439,E2 19453.439} C_VEL
LIN {X 0,Y 394.966,Z 602.688,A -85,B 0,C 180,E1 19451.756,E2 19451.756} C_VEL
LIN {X 0,Y 394.369,Z 612.812,A -85,B 0,C 180,E1 19450.073,E2 19450.073} C_VEL
LIN {X 0,Y 393.922,Z 621.273,A -85,B 0,C 180,E1 19448.316,E2 19448.316} C_VEL
LIN {X 0,Y 393.587,Z 628.822,A -85,B 0,C 180,E1 19446.269,E2 19446.269} C_VEL
LIN {X 0,Y 393.429,Z 634.035,A -85,B 0,C 180,E1 19444.37,E2 19444.37} C_VEL
LIN {X 0,Y 393.387,Z 638.066,A -85,B 0,C 180,E1 19442.183,E2 19442.183} C_VEL
LIN {X 0,Y 393.472,Z 640.042,A -85,B 0,C 180,E1 19440.144,E2 19440.144} C_VEL
LIN {X 0,Y 393.693,Z 640.354,A -85,B 0,C 180,E1 19437.96,E2 19437.96} C_VEL
LIN {X 0,Y 394.05,Z 638.689,A -85,B 0,C 180,E1 19435.778,E2 19435.778} C_VEL
LIN {X 0,Y 394.55,Z 635.401,A -85,B 0,C 180,E1 19433.742,E2 19433.742} C_VEL
LIN {X 0,Y 395.223,Z 630.199,A -85,B 0,C 180,E1 19431.707,E2 19431.707} C_VEL
LIN {X 0,Y 396.054,Z 623.537,A -85,B 0,C 180,E1 19429.819,E2 19429.819} C_VEL
LIN {X 0,Y 397.11,Z 614.805,A -85,B 0,C 180,E1 19427.936,E2 19427.936} C_VEL
LIN {X 0,Y 398.279,Z 604.418,A -85,B 0,C 180,E1 19426.201,E2 19426.201} C_VEL
LIN {X 0,Y 399.524,Z 592.399,A -85,B 0,C 180,E1 19424.615,E2 19424.615} C_VEL
LIN {X 0,Y 400.861,Z 578.641,A -85,B 0,C 180,E1 19423.18,E2 19423.18} C_VEL
LIN {X 0,Y 402.118,Z 563.568,A -85,B 0,C 180,E1 19421.965,E2 19421.965} C_VEL
LIN {X 0,Y 403.318,Z 546.504,A -85,B 0,C 180,E1 19420.935,E2 19420.935} C_VEL
LIN {X 0,Y 404.327,Z 528.498,A -85,B 0,C 180,E1 19420.172,E2 19420.172} C_VEL
LIN {X 0,Y 411.338,Z 439.177,A -85,B 0,C 180,E1 19417.224,E2 19417.224} C_VEL
LIN {X 0,Y 411.651,Z 433.14,A -85,B 0,C 180,E1 19416.995,E2 19416.995} C_VEL
LIN {X 0,Y 408.936,Z 414.676,A -85,B 0,C 180,E1 19415.815,E2 19415.815} C_VEL
LIN {X 0,Y 406.671,Z 402.484,A -85,B 0,C 180,E1 19414.904,E2 19414.904} C_VEL
LIN {X 0,Y 411.24,Z 379.25,A -85,B 0,C 180,E1 19410.903,E2 19410.903} C_VEL
LIN {X 0,Y 416.287,Z 359.629,A -85,B 0,C 180,E1 19407.287,E2 19407.287} C_VEL
LIN {X 0,Y 415.357,Z 352.667,A -85,B 0,C 180,E1 19405.044,E2 19405.044} C_VEL
LIN {X 0,Y 414.522,Z 347.62,A -85,B 0,C 180,E1 19402.912,E2 19402.912} C_VEL
LIN {X 0,Y 413.889,Z 344.327,A -85,B 0,C 180,E1 19400.91,E2 19400.91} C_VEL
LIN {X 0,Y 413.714,Z 343.064,A -85,B 0,C 180,E1 19399.793,E2 19399.793} C_VEL
LIN {X 0,Y 413.771,Z 341.818,A -85,B 0,C 180,E1 19397.231,E2 19397.231} C_VEL
LIN {X 0,Y 414.118,Z 342.611,A -85,B 0,C 180,E1 19395.363,E2 19395.363} C_VEL
LIN {X 0,Y 415.254,Z 345.062,A -85,B 0,C 180,E1 19393.144,E2 19393.144} C_VEL
LIN {X 0,Y 416.589,Z 349.376,A -85,B 0,C 180,E1 19391.092,E2 19391.092} C_VEL
LIN {X 0,Y 418.257,Z 355.199,A -85,B 0,C 180,E1 19389.133,E2 19389.133} C_VEL
LIN {X 0,Y 419.426,Z 360.386,A -85,B 0,C 180,E1 19387.783,E2 19387.783} C_VEL
LIN {X 0,Y 413.389,Z 383.432,A -85,B 0,C 180,E1 19384.808,E2 19384.808} C_VEL
LIN {X 0,Y 411.424,Z 393.701,A -85,B 0,C 180,E1 19383.594,E2 19383.594} C_VEL
LIN {X 0,Y 413.082,Z 409.418,A -85,B 0,C 180,E1 19382.858,E2 19382.858} C_VEL
LIN {X 0,Y 413.198,Z 417.031,A -85,B 0,C 180,E1 19382.597,E2 19382.597} C_VEL
LIN {X 0,Y 408.673,Z 508.972,A -85,B 0,C 180,E1 19380.366,E2 19380.366} C_VEL
LIN {X 0,Y 405.852,Z 584.93,A -85,B 0,C 180,E1 19378.647,E2 19378.647} C_VEL
LIN {X 0,Y 404.476,Z 604.284,A -85,B 0,C 180,E1 19377.956,E2 19377.956} C_VEL
LIN {X 0,Y 402.836,Z 622.92,A -85,B 0,C 180,E1 19377.015,E2 19377.015} C_VEL
LIN {X 0,Y 400.994,Z 641.128,A -85,B 0,C 180,E1 19375.793,E2 19375.793} C_VEL
LIN {X 0,Y 399.142,Z 658.276,A -85,B 0,C 180,E1 19374.336,E2 19374.336} C_VEL
LIN {X 0,Y 397.358,Z 674.455,A -85,B 0,C 180,E1 19372.644,E2 19372.644} C_VEL
LIN {X 0,Y 395.765,Z 689.617,A -85,B 0,C 180,E1 19370.715,E2 19370.715} C_VEL
LIN {X 0,Y 394.465,Z 703.201,A -85,B 0,C 180,E1 19368.626,E2 19368.626} C_VEL
LIN {X 0,Y 393.482,Z 715.297,A -85,B 0,C 180,E1 19366.384,E2 19366.384} C_VEL
LIN {X 0,Y 392.867,Z 725.889,A -85,B 0,C 180,E1 19363.993,E2 19363.993} C_VEL
LIN {X 0,Y 392.567,Z 734.931,A -85,B 0,C 180,E1 19361.46,E2 19361.46} C_VEL
LIN {X 0,Y 392.563,Z 742,A -85,B 0,C 180,E1 19358.939,E2 19358.939} C_VEL
LIN {X 0,Y 392.693,Z 747.246,A -85,B 0,C 180,E1 19356.433,E2 19356.433} C_VEL
LIN {X 0,Y 392.882,Z 750.775,A -85,B 0,C 180,E1 19353.941,E2 19353.941} C_VEL
LIN {X 0,Y 393.014,Z 752.639,A -85,B 0,C 180,E1 19351.459,E2 19351.459} C_VEL
LIN {X 0,Y 393.023,Z 752.852,A -85,B 0,C 180,E1 19348.981,E2 19348.981} C_VEL
LIN {X 0,Y 392.892,Z 751.388,A -85,B 0,C 180,E1 19346.5,E2 19346.5} C_VEL
LIN {X 0,Y 392.705,Z 748.237,A -85,B 0,C 180,E1 19344.009,E2 19344.009} C_VEL
LIN {X 0,Y 392.56,Z 743.341,A -85,B 0,C 180,E1 19341.506,E2 19341.506} C_VEL
LIN {X 0,Y 392.55,Z 736.579,A -85,B 0,C 180,E1 19338.988,E2 19338.988} C_VEL
LIN {X 0,Y 392.802,Z 727.901,A -85,B 0,C 180,E1 19336.502,E2 19336.502} C_VEL
LIN {X 0,Y 393.325,Z 717.968,A -85,B 0,C 180,E1 19334.218,E2 19334.218} C_VEL
LIN {X 0,Y 394.153,Z 706.432,A -85,B 0,C 180,E1 19332.043,E2 19332.043} C_VEL
LIN {X 0,Y 395.294,Z 693.007,A -85,B 0,C 180,E1 19329.958,E2 19329.958} C_VEL
LIN {X 0,Y 396.648,Z 678.267,A -85,B 0,C 180,E1 19328.073,E2 19328.073} C_VEL
LIN {X 0,Y 398.114,Z 662.791,A -85,B 0,C 180,E1 19326.45,E2 19326.45} C_VEL
LIN {X 0,Y 399.586,Z 646.53,A -85,B 0,C 180,E1 19325.064,E2 19325.064} C_VEL
LIN {X 0,Y 401.024,Z 629.297,A -85,B 0,C 180,E1 19323.894,E2 19323.894} C_VEL
LIN {X 0,Y 402.363,Z 610.764,A -85,B 0,C 180,E1 19322.939,E2 19322.939} C_VEL
LIN {X 0,Y 403.418,Z 592.105,A -85,B 0,C 180,E1 19322.26,E2 19322.26} C_VEL
LIN {X 0,Y 404.085,Z 569.553,A -85,B 0,C 180,E1 19321.745,E2 19321.745} C_VEL
LIN {X 0,Y 407.815,Z 412.355,A -85,B 0,C 180,E1 19318.606,E2 19318.606} C_VEL
LIN {X 0,Y 405.331,Z 388.23,A -85,B 0,C 180,E1 19317.889,E2 19317.889} C_VEL
LIN {X 0,Y 409.751,Z 348.654,A -85,B 0,C 180,E1 19313.808,E2 19313.808} C_VEL
LIN {X 0,Y 401.895,Z 325.466,A -85,B 0,C 180,E1 19310.441,E2 19310.441} C_VEL
LIN {X 0,Y 394.136,Z 304.073,A -85,B 0,C 180,E1 19307.046,E2 19307.046} C_VEL
LIN {X 0,Y 393.489,Z 301.784,A -85,B 0,C 180,E1 19306.682,E2 19306.682} C_VEL
LIN {X 0,Y 393.489,Z 301.78,A -85,B 0,C 180,E1 19302.724,E2 19302.724} C_VEL
LIN {X 0,Y 393.489,Z 301.781,A -85,B 0,C 180,E1 19298.69,E2 19298.69} C_VEL
LIN {X 0,Y 393.491,Z 301.778,A -85,B 0,C 180,E1 19294.695,E2 19294.695} C_VEL
LIN {X 0,Y 393.491,Z 301.778,A -85,B 0,C 180,E1 19290.715,E2 19290.715} C_VEL
LIN {X 0,Y 393.493,Z 301.778,A -85,B 0,C 180,E1 19286.73,E2 19286.73} C_VEL
LIN {X 0,Y 393.494,Z 301.778,A -85,B 0,C 180,E1 19282.722,E2 19282.722} C_VEL
LIN {X 0,Y 393.495,Z 301.778,A -85,B 0,C 180,E1 19278.674,E2 19278.674} C_VEL
LIN {X 0,Y 393.494,Z 301.778,A -85,B 0,C 180,E1 19274.722,E2 19274.722} C_VEL
LIN {X 0,Y 393.499,Z 301.778,A -85,B 0,C 180,E1 19270.84,E2 19270.84} C_VEL
LIN {X 0,Y 393.507,Z 301.777,A -85,B 0,C 180,E1 19267.007,E2 19267.007} C_VEL
LIN {X 0,Y 393.514,Z 301.777,A -85,B 0,C 180,E1 19263.109,E2 19263.109} C_VEL
LIN {X 0,Y 393.53,Z 301.777,A -85,B 0,C 180,E1 19259.274,E2 19259.274} C_VEL
LIN {X 0,Y 393.533,Z 301.777,A -85,B 0,C 180,E1 19255.339,E2 19255.339} C_VEL
LIN {X 0,Y 393.544,Z 301.776,A -85,B 0,C 180,E1 19251.381,E2 19251.381} C_VEL
LIN {X 0,Y 393.54,Z 301.776,A -85,B 0,C 180,E1 19247.316,E2 19247.316} C_VEL
LIN {X 0,Y 393.549,Z 301.777,A -85,B 0,C 180,E1 19243.471,E2 19243.471} C_VEL
LIN {X 0,Y 393.553,Z 301.777,A -85,B 0,C 180,E1 19239.479,E2 19239.479} C_VEL
LIN {X 0,Y 393.548,Z 301.778,A -85,B 0,C 180,E1 19235.539,E2 19235.539} C_VEL
LIN {X 0,Y 393.558,Z 301.776,A -85,B 0,C 180,E1 19231.473,E2 19231.473} C_VEL
LIN {X 0,Y 393.554,Z 301.777,A -85,B 0,C 180,E1 19227.506,E2 19227.506} C_VEL
LIN {X 0,Y 393.549,Z 301.778,A -85,B 0,C 180,E1 19223.526,E2 19223.526} C_VEL
LIN {X 0,Y 393.548,Z 301.777,A -85,B 0,C 180,E1 19219.623,E2 19219.623} C_VEL
LIN {X 0,Y 393.538,Z 301.778,A -85,B 0,C 180,E1 19215.682,E2 19215.682} C_VEL
LIN {X 0,Y 393.541,Z 301.777,A -85,B 0,C 180,E1 19211.677,E2 19211.677} C_VEL
LIN {X 0,Y 393.53,Z 301.777,A -85,B 0,C 180,E1 19207.804,E2 19207.804} C_VEL
LIN {X 0,Y 393.531,Z 301.777,A -85,B 0,C 180,E1 19203.807,E2 19203.807} C_VEL
LIN {X 0,Y 393.524,Z 301.776,A -85,B 0,C 180,E1 19199.963,E2 19199.963} C_VEL
LIN {X 0,Y 393.521,Z 301.776,A -85,B 0,C 180,E1 19196.074,E2 19196.074} C_VEL
LIN {X 0,Y 393.516,Z 301.776,A -85,B 0,C 180,E1 19192.245,E2 19192.245} C_VEL
LIN {X 0,Y 393.519,Z 301.775,A -85,B 0,C 180,E1 19188.21,E2 19188.21} C_VEL
LIN {X 0,Y 393.518,Z 301.775,A -85,B 0,C 180,E1 19184.267,E2 19184.267} C_VEL
LIN {X 0,Y 393.518,Z 301.775,A -85,B 0,C 180,E1 19180.244,E2 19180.244} C_VEL
LIN {X 0,Y 393.52,Z 301.775,A -85,B 0,C 180,E1 19176.271,E2 19176.271} C_VEL
LIN {X 0,Y 393.52,Z 301.775,A -85,B 0,C 180,E1 19172.183,E2 19172.183} C_VEL
LIN {X 0,Y 393.521,Z 301.775,A -85,B 0,C 180,E1 19168.252,E2 19168.252} C_VEL
LIN {X 0,Y 393.523,Z 301.774,A -85,B 0,C 180,E1 19164.312,E2 19164.312} C_VEL
LIN {X 0,Y 393.525,Z 301.774,A -85,B 0,C 180,E1 19160.345,E2 19160.345} C_VEL
LIN {X 0,Y 393.526,Z 301.774,A -85,B 0,C 180,E1 19156.331,E2 19156.331} C_VEL
LIN {X 0,Y 393.53,Z 301.773,A -85,B 0,C 180,E1 19152.4,E2 19152.4} C_VEL
LIN {X 0,Y 393.537,Z 301.773,A -85,B 0,C 180,E1 19148.538,E2 19148.538} C_VEL
LIN {X 0,Y 393.531,Z 301.775,A -85,B 0,C 180,E1 19147.822,E2 19147.822} C_VEL
LIN {X 0,Y 392.588,Z 301.9,A -85,B 0,C 180,E1 19146.7,E2 19146.7} C_VEL
LIN {X 0,Y 388.026,Z 302.469,A -85,B 0,C 180,E1 19144.583,E2 19144.583} C_VEL
LIN {X 0,Y 385.775,Z 302.744,A -85,B 0,C 180,E1 19143.125,E2 19143.125} C_VEL
LIN {X 0,Y 385.613,Z 302.761,A -85,B 0,C 180,E1 19142.71,E2 19142.71} C_VEL
LIN {X 0,Y 385.617,Z 302.761,A -85,B 0,C 180,E1 19138.762,E2 19138.762} C_VEL
LIN {X 0,Y 385.613,Z 302.761,A -85,B 0,C 180,E1 19134.757,E2 19134.757} C_VEL
LIN {X 0,Y 385.621,Z 302.76,A -85,B 0,C 180,E1 19130.752,E2 19130.752} C_VEL
LIN {X 0,Y 385.618,Z 302.761,A -85,B 0,C 180,E1 19126.764,E2 19126.764} C_VEL
LIN {X 0,Y 385.623,Z 302.765,A -85,B 0,C 180,E1 19122.787,E2 19122.787} C_VEL
LIN {X 0,Y 385.631,Z 302.764,A -85,B 0,C 180,E1 19118.859,E2 19118.859} C_VEL
LIN {X 0,Y 385.623,Z 302.946,A -85,B 0,C 180,E1 19117.724,E2 19117.724} C_VEL
LIN {X 0,Y 390.99,Z 321.815,A -85,B 0,C 180,E1 19114.048,E2 19114.048} C_VEL
LIN {X 0,Y 395.615,Z 339.743,A -85,B 0,C 180,E1 19110.76,E2 19110.76} C_VEL
LIN {X 0,Y 393.053,Z 366.634,A -85,B 0,C 180,E1 19106.676,E2 19106.676} C_VEL
LIN {X 0,Y 390.653,Z 395.076,A -85,B 0,C 180,E1 19102.415,E2 19102.415} C_VEL
LIN {X 0,Y 390.168,Z 402.724,A -85,B 0,C 180,E1 19101.325,E2 19101.325} C_VEL
LIN {X 0,Y 393.719,Z 430.21,A -85,B 0,C 180,E1 19100.415,E2 19100.415} C_VEL
LIN {X 0,Y 390.784,Z 528.653,A -85,B 0,C 180,E1 19097.969,E2 19097.969} C_VEL
LIN {X 0,Y 390.265,Z 544.371,A -85,B 0,C 180,E1 19097.325,E2 19097.325} C_VEL
LIN {X 0,Y 389.571,Z 560.216,A -85,B 0,C 180,E1 19096.396,E2 19096.396} C_VEL
LIN {X 0,Y 388.765,Z 575.315,A -85,B 0,C 180,E1 19095.206,E2 19095.206} C_VEL
LIN {X 0,Y 387.991,Z 588.553,A -85,B 0,C 180,E1 19093.864,E2 19093.864} C_VEL
LIN {X 0,Y 387.24,Z 600.883,A -85,B 0,C 180,E1 19092.297,E2 19092.297} C_VEL
LIN {X 0,Y 386.59,Z 611.655,A -85,B 0,C 180,E1 19090.579,E2 19090.579} C_VEL
LIN {X 0,Y 386.049,Z 621.22,A -85,B 0,C 180,E1 19088.637,E2 19088.637} C_VEL
LIN {X 0,Y 385.706,Z 628.652,A -85,B 0,C 180,E1 19086.697,E2 19086.697} C_VEL
LIN {X 0,Y 385.513,Z 634.619,A -85,B 0,C 180,E1 19084.609,E2 19084.609} C_VEL
LIN {X 0,Y 385.46,Z 638.683,A -85,B 0,C 180,E1 19082.525,E2 19082.525} C_VEL
LIN {X 0,Y 385.557,Z 641.168,A -85,B 0,C 180,E1 19080.295,E2 19080.295} C_VEL
LIN {X 0,Y 385.784,Z 641.689,A -85,B 0,C 180,E1 19078.067,E2 19078.067} C_VEL
LIN {X 0,Y 386.144,Z 640.484,A -85,B 0,C 180,E1 19075.989,E2 19075.989} C_VEL
LIN {X 0,Y 386.705,Z 637.234,A -85,B 0,C 180,E1 19073.764,E2 19073.764} C_VEL
LIN {X 0,Y 387.433,Z 632.339,A -85,B 0,C 180,E1 19071.689,E2 19071.689} C_VEL
LIN {X 0,Y 388.405,Z 625.44,A -85,B 0,C 180,E1 19069.617,E2 19069.617} C_VEL
LIN {X 0,Y 389.53,Z 616.822,A -85,B 0,C 180,E1 19067.697,E2 19067.697} C_VEL
LIN {X 0,Y 390.799,Z 606.72,A -85,B 0,C 180,E1 19065.931,E2 19065.931} C_VEL
LIN {X 0,Y 392.146,Z 595.076,A -85,B 0,C 180,E1 19064.318,E2 19064.318} C_VEL
LIN {X 0,Y 393.546,Z 581.633,A -85,B 0,C 180,E1 19062.858,E2 19062.858} C_VEL
LIN {X 0,Y 394.903,Z 567.303,A -85,B 0,C 180,E1 19061.624,E2 19061.624} C_VEL
LIN {X 0,Y 396.129,Z 552.068,A -85,B 0,C 180,E1 19060.613,E2 19060.613} C_VEL
LIN {X 0,Y 397.252,Z 534.821,A -85,B 0,C 180,E1 19059.779,E2 19059.779} C_VEL
LIN {X 0,Y 403.613,Z 456.779,A -85,B 0,C 180,E1 19057.082,E2 19057.082} C_VEL
LIN {X 0,Y 405.539,Z 435.021,A -85,B 0,C 180,E1 19056.312,E2 19056.312} C_VEL
LIN {X 0,Y 402.987,Z 416.348,A -85,B 0,C 180,E1 19055.057,E2 19055.057} C_VEL
LIN {X 0,Y 400.459,Z 402.302,A -85,B 0,C 180,E1 19053.931,E2 19053.931} C_VEL
LIN {X 0,Y 405.594,Z 379.185,A -85,B 0,C 180,E1 19049.807,E2 19049.807} C_VEL
LIN {X 0,Y 410.013,Z 363.842,A -85,B 0,C 180,E1 19046.889,E2 19046.889} C_VEL
LIN {X 0,Y 409.317,Z 357.322,A -85,B 0,C 180,E1 19044.676,E2 19044.676} C_VEL
LIN {X 0,Y 408.622,Z 352.485,A -85,B 0,C 180,E1 19042.449,E2 19042.449} C_VEL
LIN {X 0,Y 408.275,Z 349.046,A -85,B 0,C 180,E1 19040.045,E2 19040.045} C_VEL
LIN {X 0,Y 408.326,Z 347.696,A -85,B 0,C 180,E1 19037.275,E2 19037.275} C_VEL
LIN {X 0,Y 408.701,Z 348.501,A -85,B 0,C 180,E1 19035.392,E2 19035.392} C_VEL
LIN {X 0,Y 409.771,Z 351.032,A -85,B 0,C 180,E1 19033.148,E2 19033.148} C_VEL
LIN {X 0,Y 411.022,Z 355.141,A -85,B 0,C 180,E1 19031.167,E2 19031.167} C_VEL
LIN {X 0,Y 412.57,Z 361.139,A -85,B 0,C 180,E1 19029.147,E2 19029.147} C_VEL
LIN {X 0,Y 413.093,Z 364.855,A -85,B 0,C 180,E1 19028.202,E2 19028.202} C_VEL
LIN {X 0,Y 406.722,Z 387.495,A -85,B 0,C 180,E1 19025.204,E2 19025.204} C_VEL
LIN {X 0,Y 405.403,Z 394.106,A -85,B 0,C 180,E1 19024.411,E2 19024.411} C_VEL
LIN {X 0,Y 407.011,Z 410.046,A -85,B 0,C 180,E1 19023.602,E2 19023.602} C_VEL
LIN {X 0,Y 407.12,Z 417.945,A -85,B 0,C 180,E1 19023.314,E2 19023.314} C_VEL
LIN {X 0,Y 402.06,Z 509.757,A -85,B 0,C 180,E1 19020.994,E2 19020.994} C_VEL
LIN {X 0,Y 398.972,Z 584.04,A -85,B 0,C 180,E1 19019.245,E2 19019.245} C_VEL
LIN {X 0,Y 397.497,Z 603.416,A -85,B 0,C 180,E1 19018.536,E2 19018.536} C_VEL
LIN {X 0,Y 395.782,Z 621.255,A -85,B 0,C 180,E1 19017.619,E2 19017.619} C_VEL
LIN {X 0,Y 393.915,Z 638.579,A -85,B 0,C 180,E1 19016.454,E2 19016.454} C_VEL
LIN {X 0,Y 391.904,Z 655.914,A -85,B 0,C 180,E1 19014.977,E2 19014.977} C_VEL
LIN {X 0,Y 389.952,Z 672.227,A -85,B 0,C 180,E1 19013.259,E2 19013.259} C_VEL
LIN {X 0,Y 388.192,Z 687.511,A -85,B 0,C 180,E1 19011.296,E2 19011.296} C_VEL
LIN {X 0,Y 386.756,Z 701.215,A -85,B 0,C 180,E1 19009.168,E2 19009.168} C_VEL
LIN {X 0,Y 385.656,Z 713.436,A -85,B 0,C 180,E1 19006.881,E2 19006.881} C_VEL
LIN {X 0,Y 384.952,Z 724.171,A -85,B 0,C 180,E1 19004.44,E2 19004.44} C_VEL
LIN {X 0,Y 384.598,Z 733.324,A -85,B 0,C 180,E1 19001.853,E2 19001.853} C_VEL
LIN {X 0,Y 384.574,Z 740.496,A -85,B 0,C 180,E1 18999.277,E2 18999.277} C_VEL
LIN {X 0,Y 384.722,Z 745.844,A -85,B 0,C 180,E1 18996.717,E2 18996.717} C_VEL
LIN {X 0,Y 384.931,Z 749.465,A -85,B 0,C 180,E1 18994.172,E2 18994.172} C_VEL
LIN {X 0,Y 385.09,Z 751.414,A -85,B 0,C 180,E1 18991.638,E2 18991.638} C_VEL
LIN {X 0,Y 385.117,Z 751.689,A -85,B 0,C 180,E1 18989.109,E2 18989.109} C_VEL
LIN {X 0,Y 384.982,Z 750.273,A -85,B 0,C 180,E1 18986.577,E2 18986.577} C_VEL
LIN {X 0,Y 384.777,Z 747.161,A -85,B 0,C 180,E1 18984.035,E2 18984.035} C_VEL
LIN {X 0,Y 384.613,Z 742.29,A -85,B 0,C 180,E1 18981.48,E2 18981.48} C_VEL
LIN {X 0,Y 384.587,Z 735.543,A -85,B 0,C 180,E1 18978.909,E2 18978.909} C_VEL
LIN {X 0,Y 384.822,Z 727.298,A -85,B 0,C 180,E1 18976.478,E2 18976.478} C_VEL
LIN {X 0,Y 385.379,Z 716.922,A -85,B 0,C 180,E1 18974.038,E2 18974.038} C_VEL
LIN {X 0,Y 386.24,Z 705.346,A -85,B 0,C 180,E1 18971.817,E2 18971.817} C_VEL
LIN {X 0,Y 387.426,Z 691.87,A -85,B 0,C 180,E1 18969.69,E2 18969.69} C_VEL
LIN {X 0,Y 388.83,Z 677.163,A -85,B 0,C 180,E1 18967.78,E2 18967.78} C_VEL
LIN {X 0,Y 390.358,Z 661.62,A -85,B 0,C 180,E1 18966.125,E2 18966.125} C_VEL
LIN {X 0,Y 391.905,Z 645.158,A -85,B 0,C 180,E1 18964.703,E2 18964.703} C_VEL
LIN {X 0,Y 393.395,Z 627.742,A -85,B 0,C 180,E1 18963.51,E2 18963.51} C_VEL
LIN {X 0,Y 394.768,Z 609.291,A -85,B 0,C 180,E1 18962.557,E2 18962.557} C_VEL
LIN {X 0,Y 395.855,Z 590.527,A -85,B 0,C 180,E1 18961.872,E2 18961.872} C_VEL
LIN {X 0,Y 396.607,Z 564.154,A -85,B 0,C 180,E1 18961.279,E2 18961.279} C_VEL
LIN {X 0,Y 400.357,Z 412.739,A -85,B 0,C 180,E1 18958.172,E2 18958.172} C_VEL
LIN {X 0,Y 397.87,Z 388.673,A -85,B 0,C 180,E1 18957.468,E2 18957.468} C_VEL
LIN {X 0,Y 402.274,Z 351.015,A -85,B 0,C 180,E1 18953.503,E2 18953.503} C_VEL
LIN {X 0,Y 394.502,Z 328.161,A -85,B 0,C 180,E1 18950.119,E2 18950.119} C_VEL
LIN {X 0,Y 387.161,Z 307.727,A -85,B 0,C 180,E1 18946.815,E2 18946.815} C_VEL
LIN {X 0,Y 385.584,Z 302.768,A -85,B 0,C 180,E1 18945.979,E2 18945.979} C_VEL
LIN {X 0,Y 385.59,Z 302.768,A -85,B 0,C 180,E1 18941.911,E2 18941.911} C_VEL
LIN {X 0,Y 385.587,Z 302.768,A -85,B 0,C 180,E1 18937.922,E2 18937.922} C_VEL
LIN {X 0,Y 385.588,Z 302.768,A -85,B 0,C 180,E1 18933.886,E2 18933.886} C_VEL
LIN {X 0,Y 385.594,Z 302.767,A -85,B 0,C 180,E1 18929.86,E2 18929.86} C_VEL
LIN {X 0,Y 385.593,Z 302.768,A -85,B 0,C 180,E1 18925.827,E2 18925.827} C_VEL
LIN {X 0,Y 385.601,Z 302.767,A -85,B 0,C 180,E1 18921.767,E2 18921.767} C_VEL
LIN {X 0,Y 385.601,Z 302.768,A -85,B 0,C 180,E1 18917.663,E2 18917.663} C_VEL
LIN {X 0,Y 385.606,Z 302.768,A -85,B 0,C 180,E1 18913.65,E2 18913.65} C_VEL
LIN {X 0,Y 385.6,Z 302.767,A -85,B 0,C 180,E1 18909.554,E2 18909.554} C_VEL
LIN {X 0,Y 385.602,Z 302.768,A -85,B 0,C 180,E1 18905.657,E2 18905.657} C_VEL
LIN {X 0,Y 385.604,Z 302.768,A -85,B 0,C 180,E1 18901.637,E2 18901.637} C_VEL
LIN {X 0,Y 385.602,Z 302.768,A -85,B 0,C 180,E1 18897.624,E2 18897.624} C_VEL
LIN {X 0,Y 385.611,Z 302.767,A -85,B 0,C 180,E1 18893.601,E2 18893.601} C_VEL
LIN {X 0,Y 385.605,Z 302.767,A -85,B 0,C 180,E1 18889.545,E2 18889.545} C_VEL
LIN {X 0,Y 385.616,Z 302.765,A -85,B 0,C 180,E1 18885.436,E2 18885.436} C_VEL
LIN {X 0,Y 385.608,Z 302.765,A -85,B 0,C 180,E1 18881.404,E2 18881.404} C_VEL
LIN {X 0,Y 385.614,Z 302.764,A -85,B 0,C 180,E1 18877.376,E2 18877.376} C_VEL
LIN {X 0,Y 385.609,Z 302.765,A -85,B 0,C 180,E1 18873.351,E2 18873.351} C_VEL
LIN {X 0,Y 385.619,Z 302.764,A -85,B 0,C 180,E1 18869.407,E2 18869.407} C_VEL
LIN {X 0,Y 385.611,Z 302.765,A -85,B 0,C 180,E1 18865.403,E2 18865.403} C_VEL
LIN {X 0,Y 385.619,Z 302.763,A -85,B 0,C 180,E1 18861.3,E2 18861.3} C_VEL
LIN {X 0,Y 385.614,Z 302.765,A -85,B 0,C 180,E1 18857.414,E2 18857.414} C_VEL
LIN {X 0,Y 385.613,Z 302.765,A -85,B 0,C 180,E1 18853.401,E2 18853.401} C_VEL
LIN {X 0,Y 385.625,Z 302.764,A -85,B 0,C 180,E1 18849.411,E2 18849.411} C_VEL
LIN {X 0,Y 385.612,Z 302.765,A -85,B 0,C 180,E1 18845.324,E2 18845.324} C_VEL
LIN {X 0,Y 385.621,Z 302.763,A -85,B 0,C 180,E1 18841.235,E2 18841.235} C_VEL
LIN {X 0,Y 385.621,Z 302.763,A -85,B 0,C 180,E1 18837.216,E2 18837.216} C_VEL
LIN {X 0,Y 385.622,Z 302.763,A -85,B 0,C 180,E1 18833.209,E2 18833.209} C_VEL
LIN {X 0,Y 385.617,Z 302.764,A -85,B 0,C 180,E1 18829.225,E2 18829.225} C_VEL
LIN {X 0,Y 385.627,Z 302.762,A -85,B 0,C 180,E1 18825.18,E2 18825.18} C_VEL
LIN {X 0,Y 385.613,Z 302.763,A -85,B 0,C 180,E1 18821.061,E2 18821.061} C_VEL
LIN {X 0,Y 385.615,Z 302.762,A -85,B 0,C 180,E1 18816.999,E2 18816.999} C_VEL
LIN {X 0,Y 385.61,Z 302.762,A -85,B 0,C 180,E1 18812.971,E2 18812.971} C_VEL
LIN {X 0,Y 385.615,Z 302.762,A -85,B 0,C 180,E1 18808.959,E2 18808.959} C_VEL
LIN {X 0,Y 385.614,Z 302.762,A -85,B 0,C 180,E1 18804.941,E2 18804.941} C_VEL
LIN {X 0,Y 385.621,Z 302.762,A -85,B 0,C 180,E1 18801.047,E2 18801.047} C_VEL
LIN {X 0,Y 385.62,Z 302.761,A -85,B 0,C 180,E1 18796.962,E2 18796.962} C_VEL
LIN {X 0,Y 385.619,Z 302.762,A -85,B 0,C 180,E1 18792.962,E2 18792.962} C_VEL
LIN {X 0,Y 385.62,Z 302.761,A -85,B 0,C 180,E1 18788.874,E2 18788.874} C_VEL
LIN {X 0,Y 385.617,Z 302.761,A -85,B 0,C 180,E1 18784.834,E2 18784.834} C_VEL
LIN {X 0,Y 385.613,Z 302.761,A -85,B 0,C 180,E1 18782.71,E2 18782.71} C_VEL
LIN {X 0,Y 384.575,Z 302.895,A -85,B 0,C 180,E1 18781.565,E2 18781.565} C_VEL
LIN {X 0,Y 378.068,Z 303.701,A -85,B 0,C 180,E1 18778.252,E2 18778.252} C_VEL
LIN {X 0,Y 377.67,Z 303.754,A -85,B 0,C 180,E1 18777.491,E2 18777.491} C_VEL
LIN {X 0,Y 377.672,Z 303.755,A -85,B 0,C 180,E1 18773.438,E2 18773.438} C_VEL
LIN {X 0,Y 377.672,Z 303.754,A -85,B 0,C 180,E1 18769.443,E2 18769.443} C_VEL
LIN {X 0,Y 377.674,Z 303.754,A -85,B 0,C 180,E1 18765.406,E2 18765.406} C_VEL
LIN {X 0,Y 377.686,Z 303.754,A -85,B 0,C 180,E1 18761.248,E2 18761.248} C_VEL
LIN {X 0,Y 377.663,Z 303.76,A -85,B 0,C 180,E1 18758.346,E2 18758.346} C_VEL
LIN {X 0,Y 383.191,Z 323.319,A -85,B 0,C 180,E1 18754.457,E2 18754.457} C_VEL
LIN {X 0,Y 388.008,Z 341.946,A -85,B 0,C 180,E1 18750.972,E2 18750.972} C_VEL
LIN {X 0,Y 385.303,Z 369.112,A -85,B 0,C 180,E1 18746.786,E2 18746.786} C_VEL
LIN {X 0,Y 382.819,Z 397.329,A -85,B 0,C 180,E1 18742.494,E2 18742.494} C_VEL
LIN {X 0,Y 382.483,Z 402.56,A -85,B 0,C 180,E1 18741.746,E2 18741.746} C_VEL
LIN {X 0,Y 386.113,Z 431.119,A -85,B 0,C 180,E1 18740.771,E2 18740.771} C_VEL
LIN {X 0,Y 383.023,Z 529.584,A -85,B 0,C 180,E1 18738.243,E2 18738.243} C_VEL
LIN {X 0,Y 382.472,Z 545.41,A -85,B 0,C 180,E1 18737.572,E2 18737.572} C_VEL
LIN {X 0,Y 381.73,Z 561.693,A -85,B 0,C 180,E1 18736.586,E2 18736.586} C_VEL
LIN {X 0,Y 380.9,Z 576.689,A -85,B 0,C 180,E1 18735.372,E2 18735.372} C_VEL
LIN {X 0,Y 380.033,Z 591.167,A -85,B 0,C 180,E1 18733.85,E2 18733.85} C_VEL
LIN {X 0,Y 379.235,Z 603.674,A -85,B 0,C 180,E1 18732.174,E2 18732.174} C_VEL
LIN {X 0,Y 378.615,Z 613.716,A -85,B 0,C 180,E1 18730.497,E2 18730.497} C_VEL
LIN {X 0,Y 378.078,Z 623.33,A -85,B 0,C 180,E1 18728.472,E2 18728.472} C_VEL
LIN {X 0,Y 377.732,Z 630.877,A -85,B 0,C 180,E1 18726.381,E2 18726.381} C_VEL
LIN {X 0,Y 377.571,Z 636.232,A -85,B 0,C 180,E1 18724.402,E2 18724.402} C_VEL
LIN {X 0,Y 377.543,Z 640.405,A -85,B 0,C 180,E1 18722.123,E2 18722.123} C_VEL
LIN {X 0,Y 377.661,Z 642.529,A -85,B 0,C 180,E1 18719.998,E2 18719.998} C_VEL
LIN {X 0,Y 377.947,Z 642.974,A -85,B 0,C 180,E1 18717.724,E2 18717.724} C_VEL
LIN {X 0,Y 378.363,Z 641.611,A -85,B 0,C 180,E1 18715.603,E2 18715.603} C_VEL
LIN {X 0,Y 379.018,Z 638.297,A -85,B 0,C 180,E1 18713.332,E2 18713.332} C_VEL
LIN {X 0,Y 379.841,Z 633.244,A -85,B 0,C 180,E1 18711.216,E2 18711.216} C_VEL
LIN {X 0,Y 380.845,Z 626.77,A -85,B 0,C 180,E1 18709.255,E2 18709.255} C_VEL
LIN {X 0,Y 382.091,Z 618.238,A -85,B 0,C 180,E1 18707.3,E2 18707.3} C_VEL
LIN {X 0,Y 383.468,Z 608.164,A -85,B 0,C 180,E1 18705.502,E2 18705.502} C_VEL
LIN {X 0,Y 385.03,Z 595.772,A -85,B 0,C 180,E1 18703.756,E2 18703.756} C_VEL
LIN {X 0,Y 386.629,Z 581.952,A -85,B 0,C 180,E1 18702.23,E2 18702.23} C_VEL
LIN {X 0,Y 388.178,Z 566.433,A -85,B 0,C 180,E1 18700.904,E2 18700.904} C_VEL
LIN {X 0,Y 389.644,Z 549.573,A -85,B 0,C 180,E1 18699.808,E2 18699.808} C_VEL
LIN {X 0,Y 390.868,Z 531.867,A -85,B 0,C 180,E1 18698.989,E2 18698.989} C_VEL
LIN {X 0,Y 399.534,Z 438.47,A -85,B 0,C 180,E1 18695.672,E2 18695.672} C_VEL
LIN {X 0,Y 398.445,Z 427.019,A -85,B 0,C 180,E1 18694.925,E2 18694.925} C_VEL
LIN {X 0,Y 395.789,Z 409.586,A -85,B 0,C 180,E1 18693.559,E2 18693.559} C_VEL
LIN {X 0,Y 394.532,Z 401.904,A -85,B 0,C 180,E1 18692.858,E2 18692.858} C_VEL
LIN {X 0,Y 400.173,Z 379.516,A -85,B 0,C 180,E1 18688.707,E2 18688.707} C_VEL
LIN {X 0,Y 403.812,Z 368.184,A -85,B 0,C 180,E1 18686.483,E2 18686.483} C_VEL
LIN {X 0,Y 403.408,Z 362.299,A -85,B 0,C 180,E1 18684.375,E2 18684.375} C_VEL
LIN {X 0,Y 402.907,Z 357.686,A -85,B 0,C 180,E1 18682.108,E2 18682.108} C_VEL
LIN {X 0,Y 402.706,Z 354.695,A -85,B 0,C 180,E1 18679.792,E2 18679.792} C_VEL
LIN {X 0,Y 402.923,Z 353.575,A -85,B 0,C 180,E1 18677.16,E2 18677.16} C_VEL
LIN {X 0,Y 403.325,Z 354.533,A -85,B 0,C 180,E1 18675.246,E2 18675.246} C_VEL
LIN {X 0,Y 404.288,Z 356.852,A -85,B 0,C 180,E1 18673.241,E2 18673.241} C_VEL
LIN {X 0,Y 405.37,Z 360.603,A -85,B 0,C 180,E1 18671.38,E2 18671.38} C_VEL
LIN {X 0,Y 406.72,Z 366.371,A -85,B 0,C 180,E1 18669.366,E2 18669.366} C_VEL
LIN {X 0,Y 406.958,Z 368.908,A -85,B 0,C 180,E1 18668.704,E2 18668.704} C_VEL
LIN {X 0,Y 400.364,Z 390.693,A -85,B 0,C 180,E1 18665.741,E2 18665.741} C_VEL
LIN {X 0,Y 399.589,Z 394.467,A -85,B 0,C 180,E1 18665.284,E2 18665.284} C_VEL
LIN {X 0,Y 401.16,Z 410.572,A -85,B 0,C 180,E1 18664.401,E2 18664.401} C_VEL
LIN {X 0,Y 401.237,Z 418.883,A -85,B 0,C 180,E1 18664.072,E2 18664.072} C_VEL
LIN {X 0,Y 395.864,Z 505.379,A -85,B 0,C 180,E1 18661.795,E2 18661.795} C_VEL
LIN {X 0,Y 392.186,Z 583.516,A -85,B 0,C 180,E1 18659.87,E2 18659.87} C_VEL
LIN {X 0,Y 390.584,Z 602.914,A -85,B 0,C 180,E1 18659.136,E2 18659.136} C_VEL
LIN {X 0,Y 388.672,Z 621.149,A -85,B 0,C 180,E1 18658.169,E2 18658.169} C_VEL
LIN {X 0,Y 386.564,Z 639.037,A -85,B 0,C 180,E1 18656.914,E2 18656.914} C_VEL
LIN {X 0,Y 384.362,Z 656.548,A -85,B 0,C 180,E1 18655.359,E2 18655.359} C_VEL
LIN {X 0,Y 382.279,Z 672.686,A -85,B 0,C 180,E1 18653.59,E2 18653.59} C_VEL
LIN {X 0,Y 380.417,Z 687.669,A -85,B 0,C 180,E1 18651.591,E2 18651.591} C_VEL
LIN {X 0,Y 378.894,Z 701.128,A -85,B 0,C 180,E1 18649.422,E2 18649.422} C_VEL
LIN {X 0,Y 377.729,Z 713.112,A -85,B 0,C 180,E1 18647.088,E2 18647.088} C_VEL
LIN {X 0,Y 376.981,Z 723.645,A -85,B 0,C 180,E1 18644.595,E2 18644.595} C_VEL
LIN {X 0,Y 376.612,Z 732.659,A -85,B 0,C 180,E1 18641.952,E2 18641.952} C_VEL
LIN {X 0,Y 376.597,Z 739.71,A -85,B 0,C 180,E1 18639.321,E2 18639.321} C_VEL
LIN {X 0,Y 376.769,Z 744.941,A -85,B 0,C 180,E1 18636.707,E2 18636.707} C_VEL
LIN {X 0,Y 377.006,Z 748.446,A -85,B 0,C 180,E1 18634.107,E2 18634.107} C_VEL
LIN {X 0,Y 377.183,Z 750.268,A -85,B 0,C 180,E1 18631.52,E2 18631.52} C_VEL
LIN {X 0,Y 377.208,Z 750.469,A -85,B 0,C 180,E1 18629.09,E2 18629.09} C_VEL
LIN {X 0,Y 377.062,Z 749.015,A -85,B 0,C 180,E1 18626.505,E2 18626.505} C_VEL
LIN {X 0,Y 376.837,Z 745.841,A -85,B 0,C 180,E1 18623.909,E2 18623.909} C_VEL
LIN {X 0,Y 376.66,Z 740.879,A -85,B 0,C 180,E1 18621.298,E2 18621.298} C_VEL
LIN {X 0,Y 376.634,Z 733.992,A -85,B 0,C 180,E1 18618.672,E2 18618.672} C_VEL
LIN {X 0,Y 376.899,Z 725.487,A -85,B 0,C 180,E1 18616.159,E2 18616.159} C_VEL
LIN {X 0,Y 377.485,Z 715.069,A -85,B 0,C 180,E1 18613.695,E2 18613.695} C_VEL
LIN {X 0,Y 378.448,Z 702.908,A -85,B 0,C 180,E1 18611.358,E2 18611.358} C_VEL
LIN {X 0,Y 379.622,Z 690.13,A -85,B 0,C 180,E1 18609.335,E2 18609.335} C_VEL
LIN {X 0,Y 381.024,Z 675.964,A -85,B 0,C 180,E1 18607.474,E2 18607.474} C_VEL
LIN {X 0,Y 382.619,Z 660.263,A -85,B 0,C 180,E1 18605.779,E2 18605.779} C_VEL
LIN {X 0,Y 384.238,Z 643.61,A -85,B 0,C 180,E1 18604.326,E2 18604.326} C_VEL
LIN {X 0,Y 385.797,Z 625.761,A -85,B 0,C 180,E1 18603.105,E2 18603.105} C_VEL
LIN {X 0,Y 387.187,Z 607.393,A -85,B 0,C 180,E1 18602.156,E2 18602.156} C_VEL
LIN {X 0,Y 388.322,Z 587.968,A -85,B 0,C 180,E1 18601.455,E2 18601.455} C_VEL
LIN {X 0,Y 389.194,Z 555.651,A -85,B 0,C 180,E1 18600.745,E2 18600.745} C_VEL
LIN {X 0,Y 392.912,Z 413.224,A -85,B 0,C 180,E1 18597.734,E2 18597.734} C_VEL
LIN {X 0,Y 390.456,Z 388.763,A -85,B 0,C 180,E1 18597.002,E2 18597.002} C_VEL
LIN {X 0,Y 394.741,Z 353.212,A -85,B 0,C 180,E1 18593.171,E2 18593.171} C_VEL
LIN {X 0,Y 386.888,Z 330.106,A -85,B 0,C 180,E1 18589.677,E2 18589.677} C_VEL
LIN {X 0,Y 379.446,Z 309.238,A -85,B 0,C 180,E1 18586.222,E2 18586.222} C_VEL
LIN {X 0,Y 377.626,Z 303.76,A -85,B 0,C 180,E1 18585.252,E2 18585.252} C_VEL
LIN {X 0,Y 377.626,Z 303.759,A -85,B 0,C 180,E1 18581.242,E2 18581.242} C_VEL
LIN {X 0,Y 377.633,Z 303.756,A -85,B 0,C 180,E1 18577.326,E2 18577.326} C_VEL
LIN {X 0,Y 377.645,Z 303.756,A -85,B 0,C 180,E1 18573.417,E2 18573.417} C_VEL
LIN {X 0,Y 377.649,Z 303.755,A -85,B 0,C 180,E1 18569.421,E2 18569.421} C_VEL
LIN {X 0,Y 377.646,Z 303.756,A -85,B 0,C 180,E1 18565.4,E2 18565.4} C_VEL
LIN {X 0,Y 377.652,Z 303.755,A -85,B 0,C 180,E1 18561.432,E2 18561.432} C_VEL
LIN {X 0,Y 377.651,Z 303.755,A -85,B 0,C 180,E1 18557.41,E2 18557.41} C_VEL
LIN {X 0,Y 377.658,Z 303.755,A -85,B 0,C 180,E1 18553.475,E2 18553.475} C_VEL
LIN {X 0,Y 377.656,Z 303.756,A -85,B 0,C 180,E1 18549.45,E2 18549.45} C_VEL
LIN {X 0,Y 377.66,Z 303.755,A -85,B 0,C 180,E1 18545.471,E2 18545.471} C_VEL
LIN {X 0,Y 377.657,Z 303.755,A -85,B 0,C 180,E1 18541.367,E2 18541.367} C_VEL
LIN {X 0,Y 377.659,Z 303.755,A -85,B 0,C 180,E1 18537.423,E2 18537.423} C_VEL
LIN {X 0,Y 377.658,Z 303.754,A -85,B 0,C 180,E1 18533.313,E2 18533.313} C_VEL
LIN {X 0,Y 377.658,Z 303.754,A -85,B 0,C 180,E1 18529.322,E2 18529.322} C_VEL
LIN {X 0,Y 377.661,Z 303.754,A -85,B 0,C 180,E1 18525.279,E2 18525.279} C_VEL
LIN {X 0,Y 377.663,Z 303.754,A -85,B 0,C 180,E1 18521.319,E2 18521.319} C_VEL
LIN {X 0,Y 377.666,Z 303.753,A -85,B 0,C 180,E1 18517.264,E2 18517.264} C_VEL
LIN {X 0,Y 377.659,Z 303.753,A -85,B 0,C 180,E1 18513.15,E2 18513.15} C_VEL
LIN {X 0,Y 377.671,Z 303.753,A -85,B 0,C 180,E1 18509.276,E2 18509.276} C_VEL
LIN {X 0,Y 377.66,Z 303.753,A -85,B 0,C 180,E1 18505.155,E2 18505.155} C_VEL
LIN {X 0,Y 377.661,Z 303.753,A -85,B 0,C 180,E1 18501.109,E2 18501.109} C_VEL
LIN {X 0,Y 377.662,Z 303.753,A -85,B 0,C 180,E1 18497.129,E2 18497.129} C_VEL
LIN {X 0,Y 377.661,Z 303.753,A -85,B 0,C 180,E1 18493.059,E2 18493.059} C_VEL
LIN {X 0,Y 377.663,Z 303.752,A -85,B 0,C 180,E1 18489.056,E2 18489.056} C_VEL
LIN {X 0,Y 377.665,Z 303.752,A -85,B 0,C 180,E1 18485.063,E2 18485.063} C_VEL
LIN {X 0,Y 377.672,Z 303.752,A -85,B 0,C 180,E1 18481.079,E2 18481.079} C_VEL
LIN {X 0,Y 377.671,Z 303.752,A -85,B 0,C 180,E1 18477.087,E2 18477.087} C_VEL
LIN {X 0,Y 377.673,Z 303.751,A -85,B 0,C 180,E1 18473.066,E2 18473.066} C_VEL
LIN {X 0,Y 377.673,Z 303.752,A -85,B 0,C 180,E1 18469.079,E2 18469.079} C_VEL
LIN {X 0,Y 377.675,Z 303.751,A -85,B 0,C 180,E1 18465.036,E2 18465.036} C_VEL
LIN {X 0,Y 377.67,Z 303.752,A -85,B 0,C 180,E1 18460.987,E2 18460.987} C_VEL
LIN {X 0,Y 377.669,Z 303.751,A -85,B 0,C 180,E1 18456.912,E2 18456.912} C_VEL
LIN {X 0,Y 377.666,Z 303.751,A -85,B 0,C 180,E1 18452.882,E2 18452.882} C_VEL
LIN {X 0,Y 377.674,Z 303.751,A -85,B 0,C 180,E1 18448.937,E2 18448.937} C_VEL
LIN {X 0,Y 377.669,Z 303.751,A -85,B 0,C 180,E1 18444.834,E2 18444.834} C_VEL
LIN {X 0,Y 377.673,Z 303.751,A -85,B 0,C 180,E1 18440.859,E2 18440.859} C_VEL
LIN {X 0,Y 377.674,Z 303.75,A -85,B 0,C 180,E1 18436.839,E2 18436.839} C_VEL
LIN {X 0,Y 377.676,Z 303.75,A -85,B 0,C 180,E1 18432.872,E2 18432.872} C_VEL
LIN {X 0,Y 377.682,Z 303.75,A -85,B 0,C 180,E1 18428.896,E2 18428.896} C_VEL
LIN {X 0,Y 377.68,Z 303.75,A -85,B 0,C 180,E1 18424.87,E2 18424.87} C_VEL
LIN {X 0,Y 377.684,Z 303.749,A -85,B 0,C 180,E1 18420.848,E2 18420.848} C_VEL
LIN {X 0,Y 377.67,Z 303.754,A -85,B 0,C 180,E1 18417.491,E2 18417.491} C_VEL
LIN {X 0,Y 376.85,Z 303.864,A -85,B 0,C 180,E1 18416.405,E2 18416.405} C_VEL
LIN {X 0,Y 373.014,Z 304.338,A -85,B 0,C 180,E1 18414.528,E2 18414.528} C_VEL
LIN {X 0,Y 370.079,Z 304.697,A -85,B 0,C 180,E1 18412.854,E2 18412.854} C_VEL
LIN {X 0,Y 369.716,Z 304.74,A -85,B 0,C 180,E1 18412.162,E2 18412.162} C_VEL
LIN {X 0,Y 369.716,Z 304.741,A -85,B 0,C 180,E1 18408.044,E2 18408.044} C_VEL
LIN {X 0,Y 369.718,Z 304.743,A -85,B 0,C 180,E1 18403.996,E2 18403.996} C_VEL
LIN {X 0,Y 369.719,Z 304.746,A -85,B 0,C 180,E1 18399.82,E2 18399.82} C_VEL
LIN {X 0,Y 369.759,Z 304.769,A -85,B 0,C 180,E1 18398.95,E2 18398.95} C_VEL
LIN {X 0,Y 375.316,Z 324.513,A -85,B 0,C 180,E1 18394.94,E2 18394.94} C_VEL
LIN {X 0,Y 380.145,Z 343.145,A -85,B 0,C 180,E1 18391.381,E2 18391.381} C_VEL
LIN {X 0,Y 380.253,Z 345.43,A -85,B 0,C 180,E1 18390.994,E2 18390.994} C_VEL
LIN {X 0,Y 377.413,Z 372.972,A -85,B 0,C 180,E1 18386.679,E2 18386.679} C_VEL
LIN {X 0,Y 374.847,Z 401.07,A -85,B 0,C 180,E1 18382.337,E2 18382.337} C_VEL
LIN {X 0,Y 374.817,Z 402.541,A -85,B 0,C 180,E1 18382.169,E2 18382.169} C_VEL
LIN {X 0,Y 378.503,Z 432.051,A -85,B 0,C 180,E1 18381.133,E2 18381.133} C_VEL
LIN {X 0,Y 375.284,Z 530.067,A -85,B 0,C 180,E1 18378.542,E2 18378.542} C_VEL
LIN {X 0,Y 374.687,Z 546.448,A -85,B 0,C 180,E1 18377.828,E2 18377.828} C_VEL
LIN {X 0,Y 373.945,Z 562.224,A -85,B 0,C 180,E1 18376.854,E2 18376.854} C_VEL
LIN {X 0,Y 373.036,Z 578.033,A -85,B 0,C 180,E1 18375.545,E2 18375.545} C_VEL
LIN {X 0,Y 372.145,Z 592.419,A -85,B 0,C 180,E1 18373.991,E2 18373.991} C_VEL
LIN {X 0,Y 371.323,Z 604.87,A -85,B 0,C 180,E1 18372.279,E2 18372.279} C_VEL
LIN {X 0,Y 370.634,Z 615.688,A -85,B 0,C 180,E1 18370.411,E2 18370.411} C_VEL
LIN {X 0,Y 370.146,Z 624.336,A -85,B 0,C 180,E1 18368.542,E2 18368.542} C_VEL
LIN {X 0,Y 369.789,Z 632.086,A -85,B 0,C 180,E1 18366.362,E2 18366.362} C_VEL
LIN {X 0,Y 369.632,Z 637.466,A -85,B 0,C 180,E1 18364.341,E2 18364.341} C_VEL
LIN {X 0,Y 369.625,Z 641.682,A -85,B 0,C 180,E1 18362.013,E2 18362.013} C_VEL
LIN {X 0,Y 369.771,Z 643.818,A -85,B 0,C 180,E1 18359.843,E2 18359.843} C_VEL
LIN {X 0,Y 370.093,Z 644.294,A -85,B 0,C 180,E1 18357.52,E2 18357.52} C_VEL
LIN {X 0,Y 370.565,Z 642.95,A -85,B 0,C 180,E1 18355.355,E2 18355.355} C_VEL
LIN {X 0,Y 371.237,Z 639.913,A -85,B 0,C 180,E1 18353.192,E2 18353.192} C_VEL
LIN {X 0,Y 372.141,Z 635.054,A -85,B 0,C 180,E1 18351.033,E2 18351.033} C_VEL
LIN {X 0,Y 373.328,Z 628.217,A -85,B 0,C 180,E1 18348.88,E2 18348.88} C_VEL
LIN {X 0,Y 374.679,Z 619.681,A -85,B 0,C 180,E1 18346.888,E2 18346.888} C_VEL
LIN {X 0,Y 376.193,Z 609.756,A -85,B 0,C 180,E1 18345.058,E2 18345.058} C_VEL
LIN {X 0,Y 377.835,Z 597.858,A -85,B 0,C 180,E1 18343.329,E2 18343.329} C_VEL
LIN {X 0,Y 379.699,Z 583.152,A -85,B 0,C 180,E1 18341.657,E2 18341.657} C_VEL
LIN {X 0,Y 381.388,Z 567.864,A -85,B 0,C 180,E1 18340.311,E2 18340.311} C_VEL
LIN {X 0,Y 383.026,Z 550.483,A -85,B 0,C 180,E1 18339.155,E2 18339.155} C_VEL
LIN {X 0,Y 384.436,Z 532.247,A -85,B 0,C 180,E1 18338.284,E2 18338.284} C_VEL
LIN {X 0,Y 393.736,Z 439.887,A -85,B 0,C 180,E1 18334.896,E2 18334.896} C_VEL
LIN {X 0,Y 392.351,Z 425.48,A -85,B 0,C 180,E1 18333.869,E2 18333.869} C_VEL
LIN {X 0,Y 389.878,Z 408.92,A -85,B 0,C 180,E1 18332.451,E2 18332.451} C_VEL
LIN {X 0,Y 388.813,Z 401.769,A -85,B 0,C 180,E1 18331.758,E2 18331.758} C_VEL
LIN {X 0,Y 394.828,Z 380.699,A -85,B 0,C 180,E1 18327.7,E2 18327.7} C_VEL
LIN {X 0,Y 397.747,Z 372.364,A -85,B 0,C 180,E1 18325.99,E2 18325.99} C_VEL
LIN {X 0,Y 397.475,Z 366.619,A -85,B 0,C 180,E1 18323.76,E2 18323.76} C_VEL
LIN {X 0,Y 397.233,Z 362.329,A -85,B 0,C 180,E1 18321.373,E2 18321.373} C_VEL
LIN {X 0,Y 397.152,Z 360.33,A -85,B 0,C 180,E1 18319.492,E2 18319.492} C_VEL
LIN {X 0,Y 397.619,Z 359.532,A -85,B 0,C 180,E1 18316.824,E2 18316.824} C_VEL
LIN {X 0,Y 398.255,Z 361.213,A -85,B 0,C 180,E1 18314.465,E2 18314.465} C_VEL
LIN {X 0,Y 398.855,Z 362.984,A -85,B 0,C 180,E1 18313.155,E2 18313.155} C_VEL
LIN {X 0,Y 399.898,Z 366.724,A -85,B 0,C 180,E1 18311.307,E2 18311.307} C_VEL
LIN {X 0,Y 401.094,Z 372.699,A -85,B 0,C 180,E1 18309.286,E2 18309.286} C_VEL
LIN {X 0,Y 394.157,Z 393.824,A -85,B 0,C 180,E1 18306.323,E2 18306.323} C_VEL
LIN {X 0,Y 394.165,Z 396.039,A -85,B 0,C 180,E1 18306.136,E2 18306.136} C_VEL
LIN {X 0,Y 395.529,Z 411.663,A -85,B 0,C 180,E1 18305.217,E2 18305.217} C_VEL
LIN {X 0,Y 395.553,Z 420.037,A -85,B 0,C 180,E1 18304.868,E2 18304.868} C_VEL
LIN {X 0,Y 389.48,Z 507.698,A -85,B 0,C 180,E1 18302.466,E2 18302.466} C_VEL
LIN {X 0,Y 385.519,Z 583.081,A -85,B 0,C 180,E1 18300.532,E2 18300.532} C_VEL
LIN {X 0,Y 383.748,Z 602.717,A -85,B 0,C 180,E1 18299.76,E2 18299.76} C_VEL
LIN {X 0,Y 381.758,Z 620.115,A -85,B 0,C 180,E1 18298.812,E2 18298.812} C_VEL
LIN {X 0,Y 379.507,Z 637.858,A -85,B 0,C 180,E1 18297.542,E2 18297.542} C_VEL
LIN {X 0,Y 377.104,Z 655.478,A -85,B 0,C 180,E1 18295.945,E2 18295.945} C_VEL
LIN {X 0,Y 374.796,Z 671.989,A -85,B 0,C 180,E1 18294.091,E2 18294.091} C_VEL
LIN {X 0,Y 372.788,Z 686.842,A -85,B 0,C 180,E1 18292.056,E2 18292.056} C_VEL
LIN {X 0,Y 371.14,Z 700.185,A -85,B 0,C 180,E1 18289.844,E2 18289.844} C_VEL
LIN {X 0,Y 369.837,Z 712.466,A -85,B 0,C 180,E1 18287.378,E2 18287.378} C_VEL
LIN {X 0,Y 369.014,Z 723.156,A -85,B 0,C 180,E1 18284.757,E2 18284.757} C_VEL
LIN {X 0,Y 368.623,Z 732.025,A -85,B 0,C 180,E1 18282.056,E2 18282.056} C_VEL
LIN {X 0,Y 368.618,Z 738.944,A -85,B 0,C 180,E1 18279.368,E2 18279.368} C_VEL
LIN {X 0,Y 368.815,Z 744.05,A -85,B 0,C 180,E1 18276.696,E2 18276.696} C_VEL
LIN {X 0,Y 369.081,Z 747.431,A -85,B 0,C 180,E1 18274.04,E2 18274.04} C_VEL
LIN {X 0,Y 369.276,Z 749.12,A -85,B 0,C 180,E1 18271.398,E2 18271.398} C_VEL
LIN {X 0,Y 369.299,Z 749.174,A -85,B 0,C 180,E1 18268.915,E2 18268.915} C_VEL
LIN {X 0,Y 369.146,Z 747.719,A -85,B 0,C 180,E1 18266.43,E2 18266.43} C_VEL
LIN {X 0,Y 368.903,Z 744.469,A -85,B 0,C 180,E1 18263.777,E2 18263.777} C_VEL
LIN {X 0,Y 368.711,Z 739.404,A -85,B 0,C 180,E1 18261.109,E2 18261.109} C_VEL
LIN {X 0,Y 368.678,Z 732.877,A -85,B 0,C 180,E1 18258.583,E2 18258.583} C_VEL
LIN {X 0,Y 368.95,Z 724.208,A -85,B 0,C 180,E1 18255.978,E2 18255.978} C_VEL
LIN {X 0,Y 369.551,Z 713.887,A -85,B 0,C 180,E1 18253.497,E2 18253.497} C_VEL
LIN {X 0,Y 370.557,Z 701.678,A -85,B 0,C 180,E1 18251.109,E2 18251.109} C_VEL
LIN {X 0,Y 371.781,Z 688.848,A -85,B 0,C 180,E1 18249.043,E2 18249.043} C_VEL
LIN {X 0,Y 373.24,Z 674.592,A -85,B 0,C 180,E1 18247.144,E2 18247.144} C_VEL
LIN {X 0,Y 374.901,Z 658.772,A -85,B 0,C 180,E1 18245.416,E2 18245.416} C_VEL
LIN {X 0,Y 376.557,Z 642.171,A -85,B 0,C 180,E1 18243.957,E2 18243.957} C_VEL
LIN {X 0,Y 378.15,Z 624.473,A -85,B 0,C 180,E1 18242.734,E2 18242.734} C_VEL
LIN {X 0,Y 379.581,Z 605.956,A -85,B 0,C 180,E1 18241.768,E2 18241.768} C_VEL
LIN {X 0,Y 380.723,Z 586.874,A -85,B 0,C 180,E1 18241.073,E2 18241.073} C_VEL
LIN {X 0,Y 381.765,Z 548.76,A -85,B 0,C 180,E1 18240.227,E2 18240.227} C_VEL
LIN {X 0,Y 385.511,Z 414.065,A -85,B 0,C 180,E1 18237.297,E2 18237.297} C_VEL
LIN {X 0,Y 383.086,Z 388.629,A -85,B 0,C 180,E1 18236.496,E2 18236.496} C_VEL
LIN {X 0,Y 387.306,Z 355.898,A -85,B 0,C 180,E1 18232.913,E2 18232.913} C_VEL
LIN {X 0,Y 379.706,Z 333.302,A -85,B 0,C 180,E1 18229.429,E2 18229.429} C_VEL
LIN {X 0,Y 372.359,Z 312.609,A -85,B 0,C 180,E1 18225.937,E2 18225.937} C_VEL
LIN {X 0,Y 369.678,Z 304.749,A -85,B 0,C 180,E1 18224.516,E2 18224.516} C_VEL
LIN {X 0,Y 369.675,Z 304.75,A -85,B 0,C 180,E1 18220.478,E2 18220.478} C_VEL
LIN {X 0,Y 369.674,Z 304.746,A -85,B 0,C 180,E1 18216.517,E2 18216.517} C_VEL
LIN {X 0,Y 369.68,Z 304.745,A -85,B 0,C 180,E1 18212.453,E2 18212.453} C_VEL
LIN {X 0,Y 369.682,Z 304.745,A -85,B 0,C 180,E1 18208.427,E2 18208.427} C_VEL
LIN {X 0,Y 369.683,Z 304.745,A -85,B 0,C 180,E1 18204.446,E2 18204.446} C_VEL
LIN {X 0,Y 369.683,Z 304.745,A -85,B 0,C 180,E1 18200.422,E2 18200.422} C_VEL
LIN {X 0,Y 369.686,Z 304.745,A -85,B 0,C 180,E1 18196.339,E2 18196.339} C_VEL
LIN {X 0,Y 369.685,Z 304.745,A -85,B 0,C 180,E1 18192.339,E2 18192.339} C_VEL
LIN {X 0,Y 369.683,Z 304.745,A -85,B 0,C 180,E1 18188.4,E2 18188.4} C_VEL
LIN {X 0,Y 369.687,Z 304.744,A -85,B 0,C 180,E1 18184.345,E2 18184.345} C_VEL
LIN {X 0,Y 369.686,Z 304.745,A -85,B 0,C 180,E1 18180.312,E2 18180.312} C_VEL
LIN {X 0,Y 369.69,Z 304.744,A -85,B 0,C 180,E1 18176.281,E2 18176.281} C_VEL
LIN {X 0,Y 369.69,Z 304.744,A -85,B 0,C 180,E1 18172.231,E2 18172.231} C_VEL
LIN {X 0,Y 369.695,Z 304.744,A -85,B 0,C 180,E1 18168.141,E2 18168.141} C_VEL
LIN {X 0,Y 369.695,Z 304.744,A -85,B 0,C 180,E1 18164.15,E2 18164.15} C_VEL
LIN {X 0,Y 369.699,Z 304.744,A -85,B 0,C 180,E1 18160.079,E2 18160.079} C_VEL
LIN {X 0,Y 369.701,Z 304.744,A -85,B 0,C 180,E1 18156.069,E2 18156.069} C_VEL
LIN {X 0,Y 369.7,Z 304.744,A -85,B 0,C 180,E1 18152.106,E2 18152.106} C_VEL
LIN {X 0,Y 369.699,Z 304.744,A -85,B 0,C 180,E1 18148.124,E2 18148.124} C_VEL
LIN {X 0,Y 369.701,Z 304.744,A -85,B 0,C 180,E1 18144.068,E2 18144.068} C_VEL
LIN {X 0,Y 369.698,Z 304.744,A -85,B 0,C 180,E1 18140.14,E2 18140.14} C_VEL
LIN {X 0,Y 369.698,Z 304.743,A -85,B 0,C 180,E1 18136.187,E2 18136.187} C_VEL
LIN {X 0,Y 369.701,Z 304.743,A -85,B 0,C 180,E1 18132.121,E2 18132.121} C_VEL
LIN {X 0,Y 369.702,Z 304.743,A -85,B 0,C 180,E1 18128.068,E2 18128.068} C_VEL
LIN {X 0,Y 369.704,Z 304.743,A -85,B 0,C 180,E1 18124.042,E2 18124.042} C_VEL
LIN {X 0,Y 369.706,Z 304.743,A -85,B 0,C 180,E1 18120.02,E2 18120.02} C_VEL
LIN {X 0,Y 369.708,Z 304.743,A -85,B 0,C 180,E1 18115.983,E2 18115.983} C_VEL
LIN {X 0,Y 369.707,Z 304.743,A -85,B 0,C 180,E1 18111.941,E2 18111.941} C_VEL
LIN {X 0,Y 369.713,Z 304.743,A -85,B 0,C 180,E1 18107.844,E2 18107.844} C_VEL
LIN {X 0,Y 369.711,Z 304.743,A -85,B 0,C 180,E1 18103.873,E2 18103.873} C_VEL
LIN {X 0,Y 369.713,Z 304.743,A -85,B 0,C 180,E1 18099.809,E2 18099.809} C_VEL
LIN {X 0,Y 369.71,Z 304.743,A -85,B 0,C 180,E1 18095.897,E2 18095.897} C_VEL
LIN {X 0,Y 369.712,Z 304.743,A -85,B 0,C 180,E1 18091.859,E2 18091.859} C_VEL
LIN {X 0,Y 369.713,Z 304.743,A -85,B 0,C 180,E1 18087.829,E2 18087.829} C_VEL
LIN {X 0,Y 369.716,Z 304.743,A -85,B 0,C 180,E1 18083.789,E2 18083.789} C_VEL
LIN {X 0,Y 369.719,Z 304.743,A -85,B 0,C 180,E1 18079.717,E2 18079.717} C_VEL
LIN {X 0,Y 369.716,Z 304.743,A -85,B 0,C 180,E1 18075.752,E2 18075.752} C_VEL
LIN {X 0,Y 369.724,Z 304.743,A -85,B 0,C 180,E1 18071.652,E2 18071.652} C_VEL
LIN {X 0,Y 369.728,Z 304.743,A -85,B 0,C 180,E1 18067.584,E2 18067.584} C_VEL
LIN {X 0,Y 369.732,Z 304.743,A -85,B 0,C 180,E1 18063.498,E2 18063.498} C_VEL
LIN {X 0,Y 369.736,Z 304.743,A -85,B 0,C 180,E1 18059.442,E2 18059.442} C_VEL
LIN {X 0,Y 369.741,Z 304.744,A -85,B 0,C 180,E1 18055.288,E2 18055.288} C_VEL
LIN {X 0,Y 369.716,Z 304.74,A -85,B 0,C 180,E1 18052.162,E2 18052.162} C_VEL
LIN {X 0,Y 368.731,Z 304.867,A -85,B 0,C 180,E1 18050.969,E2 18050.969} C_VEL
LIN {X 0,Y 362.171,Z 305.685,A -85,B 0,C 180,E1 18047.422,E2 18047.422} C_VEL
LIN {X 0,Y 361.798,Z 305.728,A -85,B 0,C 180,E1 18046.716,E2 18046.716} C_VEL
LIN {X 0,Y 361.797,Z 305.732,A -85,B 0,C 180,E1 18042.612,E2 18042.612} C_VEL
LIN {X 0,Y 361.813,Z 305.902,A -85,B 0,C 180,E1 18039.554,E2 18039.554} C_VEL
LIN {X 0,Y 367.06,Z 324.201,A -85,B 0,C 180,E1 18035.732,E2 18035.732} C_VEL
LIN {X 0,Y 371.804,Z 342.374,A -85,B 0,C 180,E1 18032.169,E2 18032.169} C_VEL
LIN {X 0,Y 372.721,Z 346.704,A -85,B 0,C 180,E1 18031.357,E2 18031.357} C_VEL
LIN {X 0,Y 369.78,Z 374.009,A -85,B 0,C 180,E1 18027.014,E2 18027.014} C_VEL
LIN {X 0,Y 367.121,Z 402.021,A -85,B 0,C 180,E1 18022.624,E2 18022.624} C_VEL
LIN {X 0,Y 370.91,Z 432.91,A -85,B 0,C 180,E1 18021.511,E2 18021.511} C_VEL
LIN {X 0,Y 367.536,Z 530.437,A -85,B 0,C 180,E1 18018.845,E2 18018.845} C_VEL
LIN {X 0,Y 366.932,Z 546.441,A -85,B 0,C 180,E1 18018.136,E2 18018.136} C_VEL
LIN {X 0,Y 366.121,Z 563.052,A -85,B 0,C 180,E1 18017.089,E2 18017.089} C_VEL
LIN {X 0,Y 365.216,Z 578.299,A -85,B 0,C 180,E1 18015.805,E2 18015.805} C_VEL
LIN {X 0,Y 364.29,Z 592.848,A -85,B 0,C 180,E1 18014.218,E2 18014.218} C_VEL
LIN {X 0,Y 363.438,Z 605.457,A -85,B 0,C 180,E1 18012.469,E2 18012.469} C_VEL
LIN {X 0,Y 362.751,Z 616.015,A -85,B 0,C 180,E1 18010.64,E2 18010.64} C_VEL
LIN {X 0,Y 362.204,Z 625.507,A -85,B 0,C 180,E1 18008.57,E2 18008.57} C_VEL
LIN {X 0,Y 361.846,Z 633.305,A -85,B 0,C 180,E1 18006.343,E2 18006.343} C_VEL
LIN {X 0,Y 361.686,Z 639.037,A -85,B 0,C 180,E1 18004.119,E2 18004.119} C_VEL
LIN {X 0,Y 361.713,Z 643.163,A -85,B 0,C 180,E1 18001.74,E2 18001.74} C_VEL
LIN {X 0,Y 361.915,Z 645.29,A -85,B 0,C 180,E1 17999.365,E2 17999.365} C_VEL
LIN {X 0,Y 362.278,Z 645.58,A -85,B 0,C 180,E1 17997.15,E2 17997.15} C_VEL
LIN {X 0,Y 362.871,Z 643.982,A -85,B 0,C 180,E1 17994.781,E2 17994.781} C_VEL
LIN {X 0,Y 363.661,Z 640.751,A -85,B 0,C 180,E1 17992.573,E2 17992.573} C_VEL
LIN {X 0,Y 364.792,Z 635.225,A -85,B 0,C 180,E1 17990.214,E2 17990.214} C_VEL
LIN {X 0,Y 366.152,Z 627.933,A -85,B 0,C 180,E1 17988.02,E2 17988.02} C_VEL
LIN {X 0,Y 367.591,Z 619.839,A -85,B 0,C 180,E1 17986.149,E2 17986.149} C_VEL
LIN {X 0,Y 369.409,Z 608.59,A -85,B 0,C 180,E1 17984.133,E2 17984.133} C_VEL
LIN {X 0,Y 371.186,Z 596.64,A -85,B 0,C 180,E1 17982.439,E2 17982.439} C_VEL
LIN {X 0,Y 372.94,Z 583.778,A -85,B 0,C 180,E1 17980.988,E2 17980.988} C_VEL
LIN {X 0,Y 374.794,Z 568.615,A -85,B 0,C 180,E1 17979.624,E2 17979.624} C_VEL
LIN {X 0,Y 376.497,Z 552.153,A -85,B 0,C 180,E1 17978.499,E2 17978.499} C_VEL
LIN {X 0,Y 378.107,Z 533.251,A -85,B 0,C 180,E1 17977.564,E2 17977.564} C_VEL
LIN {X 0,Y 388.119,Z 440.375,A -85,B 0,C 180,E1 17974.015,E2 17974.015} C_VEL
LIN {X 0,Y 386.183,Z 421.506,A -85,B 0,C 180,E1 17972.525,E2 17972.525} C_VEL
LIN {X 0,Y 383.66,Z 403.993,A -85,B 0,C 180,E1 17970.816,E2 17970.816} C_VEL
LIN {X 0,Y 383.441,Z 401.376,A -85,B 0,C 180,E1 17970.514,E2 17970.514} C_VEL
LIN {X 0,Y 389.682,Z 382.241,A -85,B 0,C 180,E1 17966.694,E2 17966.694} C_VEL
LIN {X 0,Y 391.762,Z 376.679,A -85,B 0,C 180,E1 17965.486,E2 17965.486} C_VEL
LIN {X 0,Y 391.663,Z 371.088,A -85,B 0,C 180,E1 17963.134,E2 17963.134} C_VEL
LIN {X 0,Y 391.591,Z 367.583,A -85,B 0,C 180,E1 17960.899,E2 17960.899} C_VEL
LIN {X 0,Y 391.685,Z 366.094,A -85,B 0,C 180,E1 17959.303,E2 17959.303} C_VEL
LIN {X 0,Y 392.218,Z 365.434,A -85,B 0,C 180,E1 17956.811,E2 17956.811} C_VEL
LIN {X 0,Y 393.002,Z 367.446,A -85,B 0,C 180,E1 17954.154,E2 17954.154} C_VEL
LIN {X 0,Y 394.058,Z 371.435,A -85,B 0,C 180,E1 17951.862,E2 17951.862} C_VEL
LIN {X 0,Y 395.12,Z 376.82,A -85,B 0,C 180,E1 17949.868,E2 17949.868} C_VEL
LIN {X 0,Y 388.716,Z 394.936,A -85,B 0,C 180,E1 17947.224,E2 17947.224} C_VEL
LIN {X 0,Y 390.068,Z 410.838,A -85,B 0,C 180,E1 17946.189,E2 17946.189} C_VEL
LIN {X 0,Y 390.129,Z 420.823,A -85,B 0,C 180,E1 17945.718,E2 17945.718} C_VEL
LIN {X 0,Y 383.732,Z 502.978,A -85,B 0,C 180,E1 17943.376,E2 17943.376} C_VEL
LIN {X 0,Y 378.993,Z 582.529,A -85,B 0,C 180,E1 17941.239,E2 17941.239} C_VEL
LIN {X 0,Y 377.129,Z 601.564,A -85,B 0,C 180,E1 17940.469,E2 17940.469} C_VEL
LIN {X 0,Y 374.908,Z 619.526,A -85,B 0,C 180,E1 17939.466,E2 17939.466} C_VEL
LIN {X 0,Y 372.441,Z 637.421,A -85,B 0,C 180,E1 17938.147,E2 17938.147} C_VEL
LIN {X 0,Y 369.848,Z 654.978,A -85,B 0,C 180,E1 17936.51,E2 17936.51} C_VEL
LIN {X 0,Y 367.451,Z 670.79,A -85,B 0,C 180,E1 17934.69,E2 17934.69} C_VEL
LIN {X 0,Y 365.272,Z 685.582,A -85,B 0,C 180,E1 17932.619,E2 17932.619} C_VEL
LIN {X 0,Y 363.416,Z 699.309,A -85,B 0,C 180,E1 17930.284,E2 17930.284} C_VEL
LIN {X 0,Y 362.031,Z 711.132,A -85,B 0,C 180,E1 17927.853,E2 17927.853} C_VEL
LIN {X 0,Y 361.125,Z 721.554,A -85,B 0,C 180,E1 17925.251,E2 17925.251} C_VEL
LIN {X 0,Y 360.661,Z 730.492,A -85,B 0,C 180,E1 17922.489,E2 17922.489} C_VEL
LIN {X 0,Y 360.63,Z 737.842,A -85,B 0,C 180,E1 17919.577,E2 17919.577} C_VEL
LIN {X 0,Y 360.843,Z 742.918,A -85,B 0,C 180,E1 17916.844,E2 17916.844} C_VEL
LIN {X 0,Y 361.141,Z 746.268,A -85,B 0,C 180,E1 17914.129,E2 17914.129} C_VEL
LIN {X 0,Y 361.363,Z 747.92,A -85,B 0,C 180,E1 17911.428,E2 17911.428} C_VEL
LIN {X 0,Y 361.394,Z 747.922,A -85,B 0,C 180,E1 17908.892,E2 17908.892} C_VEL
LIN {X 0,Y 361.233,Z 746.4,A -85,B 0,C 180,E1 17906.351,E2 17906.351} C_VEL
LIN {X 0,Y 360.983,Z 743.327,A -85,B 0,C 180,E1 17903.8,E2 17903.8} C_VEL
LIN {X 0,Y 360.768,Z 738.264,A -85,B 0,C 180,E1 17901.073,E2 17901.073} C_VEL
LIN {X 0,Y 360.725,Z 731.723,A -85,B 0,C 180,E1 17898.489,E2 17898.489} C_VEL
LIN {X 0,Y 360.988,Z 723.276,A -85,B 0,C 180,E1 17895.894,E2 17895.894} C_VEL
LIN {X 0,Y 361.569,Z 713.392,A -85,B 0,C 180,E1 17893.453,E2 17893.453} C_VEL
LIN {X 0,Y 362.588,Z 701.265,A -85,B 0,C 180,E1 17891.012,E2 17891.012} C_VEL
LIN {X 0,Y 363.892,Z 687.987,A -85,B 0,C 180,E1 17888.82,E2 17888.82} C_VEL
LIN {X 0,Y 365.452,Z 673.289,A -85,B 0,C 180,E1 17886.824,E2 17886.824} C_VEL
LIN {X 0,Y 367.155,Z 657.526,A -85,B 0,C 180,E1 17885.076,E2 17885.076} C_VEL
LIN {X 0,Y 368.909,Z 640.373,A -85,B 0,C 180,E1 17883.556,E2 17883.556} C_VEL
LIN {X 0,Y 370.52,Z 623.028,A -85,B 0,C 180,E1 17882.346,E2 17882.346} C_VEL
LIN {X 0,Y 372.023,Z 604.01,A -85,B 0,C 180,E1 17881.349,E2 17881.349} C_VEL
LIN {X 0,Y 373.151,Z 585.206,A -85,B 0,C 180,E1 17880.666,E2 17880.666} C_VEL
LIN {X 0,Y 378.092,Z 414.804,A -85,B 0,C 180,E1 17876.85,E2 17876.85} C_VEL
LIN {X 0,Y 375.67,Z 388.786,A -85,B 0,C 180,E1 17876.02,E2 17876.02} C_VEL
LIN {X 0,Y 379.804,Z 358.221,A -85,B 0,C 180,E1 17872.6,E2 17872.6} C_VEL
LIN {X 0,Y 371.81,Z 334.445,A -85,B 0,C 180,E1 17868.85,E2 17868.85} C_VEL
LIN {X 0,Y 364.522,Z 313.788,A -85,B 0,C 180,E1 17865.271,E2 17865.271} C_VEL
LIN {X 0,Y 361.773,Z 305.736,A -85,B 0,C 180,E1 17863.776,E2 17863.776} C_VEL
LIN {X 0,Y 361.781,Z 305.735,A -85,B 0,C 180,E1 17859.676,E2 17859.676} C_VEL
LIN {X 0,Y 361.766,Z 305.734,A -85,B 0,C 180,E1 17855.481,E2 17855.481} C_VEL
LIN {X 0,Y 361.761,Z 305.734,A -85,B 0,C 180,E1 17851.35,E2 17851.35} C_VEL
LIN {X 0,Y 361.76,Z 305.734,A -85,B 0,C 180,E1 17847.312,E2 17847.312} C_VEL
LIN {X 0,Y 361.76,Z 305.734,A -85,B 0,C 180,E1 17843.282,E2 17843.282} C_VEL
LIN {X 0,Y 361.759,Z 305.733,A -85,B 0,C 180,E1 17839.204,E2 17839.204} C_VEL
LIN {X 0,Y 361.761,Z 305.733,A -85,B 0,C 180,E1 17835.224,E2 17835.224} C_VEL
LIN {X 0,Y 361.757,Z 305.733,A -85,B 0,C 180,E1 17831.14,E2 17831.14} C_VEL
LIN {X 0,Y 361.76,Z 305.733,A -85,B 0,C 180,E1 17827.147,E2 17827.147} C_VEL
LIN {X 0,Y 361.754,Z 305.733,A -85,B 0,C 180,E1 17823.012,E2 17823.012} C_VEL
LIN {X 0,Y 361.752,Z 305.733,A -85,B 0,C 180,E1 17818.894,E2 17818.894} C_VEL
LIN {X 0,Y 361.749,Z 305.733,A -85,B 0,C 180,E1 17814.769,E2 17814.769} C_VEL
LIN {X 0,Y 361.748,Z 305.733,A -85,B 0,C 180,E1 17810.617,E2 17810.617} C_VEL
LIN {X 0,Y 361.749,Z 305.733,A -85,B 0,C 180,E1 17806.415,E2 17806.415} C_VEL
LIN {X 0,Y 361.753,Z 305.733,A -85,B 0,C 180,E1 17802.303,E2 17802.303} C_VEL
LIN {X 0,Y 361.755,Z 305.733,A -85,B 0,C 180,E1 17798.225,E2 17798.225} C_VEL
LIN {X 0,Y 361.761,Z 305.733,A -85,B 0,C 180,E1 17794.11,E2 17794.11} C_VEL
LIN {X 0,Y 361.757,Z 305.733,A -85,B 0,C 180,E1 17790.169,E2 17790.169} C_VEL
LIN {X 0,Y 361.763,Z 305.733,A -85,B 0,C 180,E1 17786.065,E2 17786.065} C_VEL
LIN {X 0,Y 361.766,Z 305.733,A -85,B 0,C 180,E1 17781.955,E2 17781.955} C_VEL
LIN {X 0,Y 361.766,Z 305.732,A -85,B 0,C 180,E1 17778.026,E2 17778.026} C_VEL
LIN {X 0,Y 361.77,Z 305.732,A -85,B 0,C 180,E1 17773.923,E2 17773.923} C_VEL
LIN {X 0,Y 361.771,Z 305.733,A -85,B 0,C 180,E1 17769.88,E2 17769.88} C_VEL
LIN {X 0,Y 361.772,Z 305.733,A -85,B 0,C 180,E1 17765.866,E2 17765.866} C_VEL
LIN {X 0,Y 361.774,Z 305.732,A -85,B 0,C 180,E1 17761.861,E2 17761.861} C_VEL
LIN {X 0,Y 361.777,Z 305.732,A -85,B 0,C 180,E1 17757.83,E2 17757.83} C_VEL
LIN {X 0,Y 361.777,Z 305.732,A -85,B 0,C 180,E1 17753.796,E2 17753.796} C_VEL
LIN {X 0,Y 361.773,Z 305.732,A -85,B 0,C 180,E1 17749.872,E2 17749.872} C_VEL
LIN {X 0,Y 361.782,Z 305.732,A -85,B 0,C 180,E1 17745.713,E2 17745.713} C_VEL
LIN {X 0,Y 361.784,Z 305.733,A -85,B 0,C 180,E1 17741.638,E2 17741.638} C_VEL
LIN {X 0,Y 361.797,Z 305.733,A -85,B 0,C 180,E1 17737.462,E2 17737.462} C_VEL
LIN {X 0,Y 361.797,Z 305.732,A -85,B 0,C 180,E1 17733.326,E2 17733.326} C_VEL
LIN {X 0,Y 361.809,Z 305.73,A -85,B 0,C 180,E1 17729.207,E2 17729.207} C_VEL
LIN {X 0,Y 361.8,Z 305.729,A -85,B 0,C 180,E1 17725.084,E2 17725.084} C_VEL
LIN {X 0,Y 361.805,Z 305.729,A -85,B 0,C 180,E1 17721.096,E2 17721.096} C_VEL
LIN {X 0,Y 361.8,Z 305.728,A -85,B 0,C 180,E1 17716.901,E2 17716.901} C_VEL
LIN {X 0,Y 361.794,Z 305.728,A -85,B 0,C 180,E1 17712.799,E2 17712.799} C_VEL
LIN {X 0,Y 361.787,Z 305.728,A -85,B 0,C 180,E1 17708.637,E2 17708.637} C_VEL
LIN {X 0,Y 361.789,Z 305.728,A -85,B 0,C 180,E1 17704.635,E2 17704.635} C_VEL
LIN {X 0,Y 361.787,Z 305.728,A -85,B 0,C 180,E1 17700.516,E2 17700.516} C_VEL
LIN {X 0,Y 361.783,Z 305.729,A -85,B 0,C 180,E1 17696.444,E2 17696.444} C_VEL
LIN {X 0,Y 361.783,Z 305.728,A -85,B 0,C 180,E1 17692.353,E2 17692.353} C_VEL
LIN {X 0,Y 361.78,Z 305.729,A -85,B 0,C 180,E1 17688.235,E2 17688.235} C_VEL
LIN {X 0,Y 361.798,Z 305.728,A -85,B 0,C 180,E1 17686.716,E2 17686.716} C_VEL
LIN {X 0,Y 360.766,Z 305.861,A -85,B 0,C 180,E1 17685.496,E2 17685.496} C_VEL
LIN {X 0,Y 354.275,Z 306.674,A -85,B 0,C 180,E1 17681.961,E2 17681.961} C_VEL
LIN {X 0,Y 353.873,Z 306.719,A -85,B 0,C 180,E1 17681.148,E2 17681.148} C_VEL
LIN {X 0,Y 353.861,Z 306.858,A -85,B 0,C 180,E1 17680.212,E2 17680.212} C_VEL
LIN {X 0,Y 359.115,Z 325.108,A -85,B 0,C 180,E1 17676.302,E2 17676.302} C_VEL
LIN {X 0,Y 363.787,Z 342.789,A -85,B 0,C 180,E1 17672.749,E2 17672.749} C_VEL
LIN {X 0,Y 365.055,Z 349.187,A -85,B 0,C 180,E1 17671.539,E2 17671.539} C_VEL
LIN {X 0,Y 361.988,Z 376.579,A -85,B 0,C 180,E1 17667.11,E2 17667.11} C_VEL
LIN {X 0,Y 359.494,Z 402.222,A -85,B 0,C 180,E1 17663.056,E2 17663.056} C_VEL
LIN {X 0,Y 363.296,Z 433.783,A -85,B 0,C 180,E1 17661.888,E2 17661.888} C_VEL
LIN {X 0,Y 359.767,Z 531.251,A -85,B 0,C 180,E1 17659.134,E2 17659.134} C_VEL
LIN {X 0,Y 359.114,Z 547.728,A -85,B 0,C 180,E1 17658.377,E2 17658.377} C_VEL
LIN {X 0,Y 358.326,Z 563.389,A -85,B 0,C 180,E1 17657.369,E2 17657.369} C_VEL
LIN {X 0,Y 357.347,Z 579.391,A -85,B 0,C 180,E1 17655.995,E2 17655.995} C_VEL
LIN {X 0,Y 356.383,Z 594.124,A -85,B 0,C 180,E1 17654.351,E2 17654.351} C_VEL
LIN {X 0,Y 355.49,Z 607.095,A -85,B 0,C 180,E1 17652.505,E2 17652.505} C_VEL
LIN {X 0,Y 354.767,Z 617.967,A -85,B 0,C 180,E1 17650.553,E2 17650.553} C_VEL
LIN {X 0,Y 354.258,Z 626.648,A -85,B 0,C 180,E1 17648.6,E2 17648.6} C_VEL
LIN {X 0,Y 353.898,Z 634.471,A -85,B 0,C 180,E1 17646.324,E2 17646.324} C_VEL
LIN {X 0,Y 353.745,Z 640.235,A -85,B 0,C 180,E1 17644.05,E2 17644.05} C_VEL
LIN {X 0,Y 353.785,Z 644.207,A -85,B 0,C 180,E1 17641.779,E2 17641.779} C_VEL
LIN {X 0,Y 354.009,Z 646.503,A -85,B 0,C 180,E1 17639.35,E2 17639.35} C_VEL
LIN {X 0,Y 354.408,Z 646.965,A -85,B 0,C 180,E1 17637.087,E2 17637.087} C_VEL
LIN {X 0,Y 355.057,Z 645.539,A -85,B 0,C 180,E1 17634.666,E2 17634.666} C_VEL
LIN {X 0,Y 355.918,Z 642.481,A -85,B 0,C 180,E1 17632.411,E2 17632.411} C_VEL
LIN {X 0,Y 357.144,Z 637.162,A -85,B 0,C 180,E1 17630.002,E2 17630.002} C_VEL
LIN {X 0,Y 358.505,Z 630.718,A -85,B 0,C 180,E1 17627.924,E2 17627.924} C_VEL
LIN {X 0,Y 360.297,Z 621.523,A -85,B 0,C 180,E1 17625.699,E2 17625.699} C_VEL
LIN {X 0,Y 362.113,Z 611.417,A -85,B 0,C 180,E1 17623.805,E2 17623.805} C_VEL
LIN {X 0,Y 364.098,Z 599.297,A -85,B 0,C 180,E1 17622.003,E2 17622.003} C_VEL
LIN {X 0,Y 366.203,Z 585.513,A -85,B 0,C 180,E1 17620.375,E2 17620.375} C_VEL
LIN {X 0,Y 368.299,Z 569.603,A -85,B 0,C 180,E1 17618.916,E2 17618.916} C_VEL
LIN {X 0,Y 370.162,Z 553.503,A -85,B 0,C 180,E1 17617.778,E2 17617.778} C_VEL
LIN {X 0,Y 371.841,Z 535.645,A -85,B 0,C 180,E1 17616.857,E2 17616.857} C_VEL
LIN {X 0,Y 382.715,Z 442.282,A -85,B 0,C 180,E1 17613.17,E2 17613.17} C_VEL
LIN {X 0,Y 381.13,Z 424.096,A -85,B 0,C 180,E1 17611.66,E2 17611.66} C_VEL
LIN {X 0,Y 379.04,Z 407.219,A -85,B 0,C 180,E1 17609.941,E2 17609.941} C_VEL
LIN {X 0,Y 378.353,Z 401.278,A -85,B 0,C 180,E1 17609.244,E2 17609.244} C_VEL
LIN {X 0,Y 385.642,Z 382.003,A -85,B 0,C 180,E1 17605.22,E2 17605.22} C_VEL
LIN {X 0,Y 385.912,Z 379.988,A -85,B 0,C 180,E1 17604.522,E2 17604.522} C_VEL
LIN {X 0,Y 386.006,Z 375.233,A -85,B 0,C 180,E1 17602.19,E2 17602.19} C_VEL
LIN {X 0,Y 386.229,Z 372.235,A -85,B 0,C 180,E1 17599.792,E2 17599.792} C_VEL
LIN {X 0,Y 386.791,Z 371.319,A -85,B 0,C 180,E1 17596.963,E2 17596.963} C_VEL
LIN {X 0,Y 387.347,Z 372.778,A -85,B 0,C 180,E1 17594.775,E2 17594.775} C_VEL
LIN {X 0,Y 387.882,Z 374.393,A -85,B 0,C 180,E1 17593.493,E2 17593.493} C_VEL
LIN {X 0,Y 388.644,Z 377.693,A -85,B 0,C 180,E1 17591.746,E2 17591.746} C_VEL
LIN {X 0,Y 389.193,Z 381.468,A -85,B 0,C 180,E1 17590.347,E2 17590.347} C_VEL
LIN {X 0,Y 383.785,Z 395.805,A -85,B 0,C 180,E1 17588.242,E2 17588.242} C_VEL
LIN {X 0,Y 384.918,Z 411.401,A -85,B 0,C 180,E1 17587.143,E2 17587.143} C_VEL
LIN {X 0,Y 384.975,Z 421.643,A -85,B 0,C 180,E1 17586.614,E2 17586.614} C_VEL
LIN {X 0,Y 377.675,Z 505.826,A -85,B 0,C 180,E1 17584.121,E2 17584.121} C_VEL
LIN {X 0,Y 372.649,Z 581.656,A -85,B 0,C 180,E1 17582.001,E2 17582.001} C_VEL
LIN {X 0,Y 370.601,Z 600.926,A -85,B 0,C 180,E1 17581.2,E2 17581.2} C_VEL
LIN {X 0,Y 368.173,Z 618.957,A -85,B 0,C 180,E1 17580.161,E2 17580.161} C_VEL
LIN {X 0,Y 365.602,Z 636.176,A -85,B 0,C 180,E1 17578.863,E2 17578.863} C_VEL
LIN {X 0,Y 362.835,Z 653.456,A -85,B 0,C 180,E1 17577.223,E2 17577.223} C_VEL
LIN {X 0,Y 360.27,Z 669.109,A -85,B 0,C 180,E1 17575.392,E2 17575.392} C_VEL
LIN {X 0,Y 357.888,Z 683.912,A -85,B 0,C 180,E1 17573.287,E2 17573.287} C_VEL
LIN {X 0,Y 355.841,Z 697.676,A -85,B 0,C 180,E1 17570.908,E2 17570.908} C_VEL
LIN {X 0,Y 354.296,Z 709.529,A -85,B 0,C 180,E1 17568.427,E2 17568.427} C_VEL
LIN {X 0,Y 353.252,Z 719.993,A -85,B 0,C 180,E1 17565.768,E2 17565.768} C_VEL
LIN {X 0,Y 352.708,Z 728.986,A -85,B 0,C 180,E1 17562.942,E2 17562.942} C_VEL
LIN {X 0,Y 352.631,Z 736.399,A -85,B 0,C 180,E1 17559.961,E2 17559.961} C_VEL
LIN {X 0,Y 352.849,Z 741.54,A -85,B 0,C 180,E1 17557.164,E2 17557.164} C_VEL
LIN {X 0,Y 353.186,Z 744.953,A -85,B 0,C 180,E1 17554.385,E2 17554.385} C_VEL
LIN {X 0,Y 353.44,Z 746.664,A -85,B 0,C 180,E1 17551.622,E2 17551.622} C_VEL
LIN {X 0,Y 353.497,Z 746.711,A -85,B 0,C 180,E1 17549.029,E2 17549.029} C_VEL
LIN {X 0,Y 353.334,Z 745.214,A -85,B 0,C 180,E1 17546.432,E2 17546.432} C_VEL
LIN {X 0,Y 353.062,Z 742.016,A -85,B 0,C 180,E1 17543.74,E2 17543.74} C_VEL
LIN {X 0,Y 352.829,Z 737.081,A -85,B 0,C 180,E1 17541.035,E2 17541.035} C_VEL
LIN {X 0,Y 352.775,Z 730.522,A -85,B 0,C 180,E1 17538.392,E2 17538.392} C_VEL
LIN {X 0,Y 353.04,Z 722.039,A -85,B 0,C 180,E1 17535.737,E2 17535.737} C_VEL
LIN {X 0,Y 353.646,Z 712.098,A -85,B 0,C 180,E1 17533.24,E2 17533.24} C_VEL
LIN {X 0,Y 354.708,Z 699.893,A -85,B 0,C 180,E1 17530.745,E2 17530.745} C_VEL
LIN {X 0,Y 356.067,Z 686.514,A -85,B 0,C 180,E1 17528.504,E2 17528.504} C_VEL
LIN {X 0,Y 357.715,Z 671.506,A -85,B 0,C 180,E1 17526.442,E2 17526.442} C_VEL
LIN {X 0,Y 359.51,Z 655.273,A -85,B 0,C 180,E1 17524.642,E2 17524.642} C_VEL
LIN {X 0,Y 361.225,Z 638.938,A -85,B 0,C 180,E1 17523.182,E2 17523.182} C_VEL
LIN {X 0,Y 362.966,Z 620.628,A -85,B 0,C 180,E1 17521.899,E2 17521.899} C_VEL
LIN {X 0,Y 364.459,Z 602.191,A -85,B 0,C 180,E1 17520.934,E2 17520.934} C_VEL
LIN {X 0,Y 365.592,Z 583.04,A -85,B 0,C 180,E1 17520.24,E2 17520.24} C_VEL
LIN {X 0,Y 370.698,Z 415.796,A -85,B 0,C 180,E1 17516.404,E2 17516.404} C_VEL
LIN {X 0,Y 368.279,Z 388.928,A -85,B 0,C 180,E1 17515.525,E2 17515.525} C_VEL
LIN {X 0,Y 372.131,Z 360.149,A -85,B 0,C 180,E1 17512.224,E2 17512.224} C_VEL
LIN {X 0,Y 364.75,Z 337.993,A -85,B 0,C 180,E1 17508.654,E2 17508.654} C_VEL
LIN {X 0,Y 357.54,Z 317.426,A -85,B 0,C 180,E1 17505.035,E2 17505.035} C_VEL
LIN {X 0,Y 353.801,Z 306.725,A -85,B 0,C 180,E1 17502.98,E2 17502.98} C_VEL
LIN {X 0,Y 353.797,Z 306.727,A -85,B 0,C 180,E1 17498.742,E2 17498.742} C_VEL
LIN {X 0,Y 353.799,Z 306.723,A -85,B 0,C 180,E1 17494.616,E2 17494.616} C_VEL
LIN {X 0,Y 353.801,Z 306.723,A -85,B 0,C 180,E1 17490.467,E2 17490.467} C_VEL
LIN {X 0,Y 353.807,Z 306.723,A -85,B 0,C 180,E1 17486.341,E2 17486.341} C_VEL
LIN {X 0,Y 353.81,Z 306.723,A -85,B 0,C 180,E1 17482.254,E2 17482.254} C_VEL
LIN {X 0,Y 353.818,Z 306.723,A -85,B 0,C 180,E1 17478.112,E2 17478.112} C_VEL
LIN {X 0,Y 353.82,Z 306.723,A -85,B 0,C 180,E1 17474.067,E2 17474.067} C_VEL
LIN {X 0,Y 353.828,Z 306.723,A -85,B 0,C 180,E1 17469.928,E2 17469.928} C_VEL
LIN {X 0,Y 353.834,Z 306.723,A -85,B 0,C 180,E1 17465.841,E2 17465.841} C_VEL
LIN {X 0,Y 353.845,Z 306.724,A -85,B 0,C 180,E1 17461.621,E2 17461.621} C_VEL
LIN {X 0,Y 353.843,Z 306.723,A -85,B 0,C 180,E1 17457.573,E2 17457.573} C_VEL
LIN {X 0,Y 353.844,Z 306.721,A -85,B 0,C 180,E1 17453.35,E2 17453.35} C_VEL
LIN {X 0,Y 353.835,Z 306.721,A -85,B 0,C 180,E1 17449.254,E2 17449.254} C_VEL
LIN {X 0,Y 353.83,Z 306.721,A -85,B 0,C 180,E1 17445.102,E2 17445.102} C_VEL
LIN {X 0,Y 353.829,Z 306.721,A -85,B 0,C 180,E1 17441.039,E2 17441.039} C_VEL
LIN {X 0,Y 353.823,Z 306.721,A -85,B 0,C 180,E1 17436.874,E2 17436.874} C_VEL
LIN {X 0,Y 353.82,Z 306.721,A -85,B 0,C 180,E1 17432.758,E2 17432.758} C_VEL
LIN {X 0,Y 353.818,Z 306.721,A -85,B 0,C 180,E1 17428.583,E2 17428.583} C_VEL
LIN {X 0,Y 353.817,Z 306.721,A -85,B 0,C 180,E1 17424.403,E2 17424.403} C_VEL
LIN {X 0,Y 353.818,Z 306.721,A -85,B 0,C 180,E1 17420.23,E2 17420.23} C_VEL
LIN {X 0,Y 353.823,Z 306.721,A -85,B 0,C 180,E1 17416.102,E2 17416.102} C_VEL
LIN {X 0,Y 353.827,Z 306.721,A -85,B 0,C 180,E1 17412.001,E2 17412.001} C_VEL
LIN {X 0,Y 353.828,Z 306.721,A -85,B 0,C 180,E1 17407.968,E2 17407.968} C_VEL
LIN {X 0,Y 353.836,Z 306.721,A -85,B 0,C 180,E1 17403.825,E2 17403.825} C_VEL
LIN {X 0,Y 353.851,Z 306.721,A -85,B 0,C 180,E1 17399.634,E2 17399.634} C_VEL
LIN {X 0,Y 353.856,Z 306.722,A -85,B 0,C 180,E1 17395.434,E2 17395.434} C_VEL
LIN {X 0,Y 353.865,Z 306.718,A -85,B 0,C 180,E1 17391.193,E2 17391.193} C_VEL
LIN {X 0,Y 353.845,Z 306.719,A -85,B 0,C 180,E1 17386.919,E2 17386.919} C_VEL
LIN {X 0,Y 353.847,Z 306.718,A -85,B 0,C 180,E1 17382.89,E2 17382.89} C_VEL
LIN {X 0,Y 353.841,Z 306.719,A -85,B 0,C 180,E1 17378.776,E2 17378.776} C_VEL
LIN {X 0,Y 353.837,Z 306.719,A -85,B 0,C 180,E1 17374.699,E2 17374.699} C_VEL
LIN {X 0,Y 353.833,Z 306.719,A -85,B 0,C 180,E1 17370.484,E2 17370.484} C_VEL
LIN {X 0,Y 353.831,Z 306.719,A -85,B 0,C 180,E1 17366.272,E2 17366.272} C_VEL
LIN {X 0,Y 353.83,Z 306.72,A -85,B 0,C 180,E1 17362.04,E2 17362.04} C_VEL
LIN {X 0,Y 353.836,Z 306.72,A -85,B 0,C 180,E1 17357.865,E2 17357.865} C_VEL
LIN {X 0,Y 353.84,Z 306.72,A -85,B 0,C 180,E1 17353.754,E2 17353.754} C_VEL
LIN {X 0,Y 353.845,Z 306.721,A -85,B 0,C 180,E1 17349.661,E2 17349.661} C_VEL
LIN {X 0,Y 353.846,Z 306.721,A -85,B 0,C 180,E1 17345.634,E2 17345.634} C_VEL
LIN {X 0,Y 353.857,Z 306.721,A -85,B 0,C 180,E1 17341.475,E2 17341.475} C_VEL
LIN {X 0,Y 353.861,Z 306.722,A -85,B 0,C 180,E1 17337.337,E2 17337.337} C_VEL
LIN {X 0,Y 353.868,Z 306.718,A -85,B 0,C 180,E1 17333.088,E2 17333.088} C_VEL
LIN {X 0,Y 353.876,Z 306.716,A -85,B 0,C 180,E1 17328.967,E2 17328.967} C_VEL
LIN {X 0,Y 353.861,Z 306.722,A -85,B 0,C 180,E1 17324.709,E2 17324.709} C_VEL
LIN {X 0,Y 353.873,Z 306.719,A -85,B 0,C 180,E1 17321.148,E2 17321.148} C_VEL
LIN {X 0,Y 353.713,Z 307.615,A -85,B 0,C 180,E1 17320.446,E2 17320.446} C_VEL
LIN {X 0,Y 353.147,Z 310.474,A -85,B 0,C 180,E1 17319.66,E2 17319.66} C_VEL
LIN {X 0,Y 351.165,Z 323.59,A -85,B 0,C 180,E1 17317.347,E2 17317.347} C_VEL
LIN {X 0,Y 351.684,Z 327.852,A -85,B 0,C 180,E1 17316.507,E2 17316.507} C_VEL
LIN {X 0,Y 356.34,Z 345.592,A -85,B 0,C 180,E1 17312.881,E2 17312.881} C_VEL
LIN {X 0,Y 357.447,Z 351.154,A -85,B 0,C 180,E1 17311.809,E2 17311.809} C_VEL
LIN {X 0,Y 354.231,Z 378.595,A -85,B 0,C 180,E1 17307.289,E2 17307.289} C_VEL
LIN {X 0,Y 351.853,Z 402.119,A -85,B 0,C 180,E1 17303.513,E2 17303.513} C_VEL
LIN {X 0,Y 355.682,Z 434.648,A -85,B 0,C 180,E1 17302.272,E2 17302.272} C_VEL
LIN {X 0,Y 352.011,Z 531.888,A -85,B 0,C 180,E1 17299.441,E2 17299.441} C_VEL
LIN {X 0,Y 351.339,Z 548.3,A -85,B 0,C 180,E1 17298.67,E2 17298.67} C_VEL
LIN {X 0,Y 350.491,Z 564.507,A -85,B 0,C 180,E1 17297.598,E2 17297.598} C_VEL
LIN {X 0,Y 349.48,Z 580.408,A -85,B 0,C 180,E1 17296.195,E2 17296.195} C_VEL
LIN {X 0,Y 348.498,Z 594.928,A -85,B 0,C 180,E1 17294.536,E2 17294.536} C_VEL
LIN {X 0,Y 347.566,Z 608.082,A -85,B 0,C 180,E1 17292.626,E2 17292.626} C_VEL
LIN {X 0,Y 346.822,Z 618.968,A -85,B 0,C 180,E1 17290.63,E2 17290.63} C_VEL
LIN {X 0,Y 346.307,Z 627.727,A -85,B 0,C 180,E1 17288.632,E2 17288.632} C_VEL
LIN {X 0,Y 345.948,Z 635.624,A -85,B 0,C 180,E1 17286.303,E2 17286.303} C_VEL
LIN {X 0,Y 345.804,Z 641.447,A -85,B 0,C 180,E1 17283.977,E2 17283.977} C_VEL
LIN {X 0,Y 345.863,Z 645.461,A -85,B 0,C 180,E1 17281.654,E2 17281.654} C_VEL
LIN {X 0,Y 346.123,Z 647.803,A -85,B 0,C 180,E1 17279.17,E2 17279.17} C_VEL
LIN {X 0,Y 346.577,Z 648.324,A -85,B 0,C 180,E1 17276.856,E2 17276.856} C_VEL
LIN {X 0,Y 347.305,Z 646.948,A -85,B 0,C 180,E1 17274.38,E2 17274.38} C_VEL
LIN {X 0,Y 348.262,Z 643.977,A -85,B 0,C 180,E1 17272.077,E2 17272.077} C_VEL
LIN {X 0,Y 349.519,Z 639.093,A -85,B 0,C 180,E1 17269.765,E2 17269.765} C_VEL
LIN {X 0,Y 351.107,Z 632.386,A -85,B 0,C 180,E1 17267.499,E2 17267.499} C_VEL
LIN {X 0,Y 352.901,Z 624.042,A -85,B 0,C 180,E1 17265.393,E2 17265.393} C_VEL
LIN {X 0,Y 355.024,Z 613.392,A -85,B 0,C 180,E1 17263.304,E2 17263.304} C_VEL
LIN {X 0,Y 357.182,Z 601.589,A -85,B 0,C 180,E1 17261.473,E2 17261.473} C_VEL
LIN {X 0,Y 359.659,Z 586.672,A -85,B 0,C 180,E1 17259.663,E2 17259.663} C_VEL
LIN {X 0,Y 361.943,Z 571.029,A -85,B 0,C 180,E1 17258.187,E2 17258.187} C_VEL
LIN {X 0,Y 364.088,Z 554.039,A -85,B 0,C 180,E1 17256.961,E2 17256.961} C_VEL
LIN {X 0,Y 366.022,Z 535.484,A -85,B 0,C 180,E1 17255.986,E2 17255.986} C_VEL
LIN {X 0,Y 377.509,Z 444.257,A -85,B 0,C 180,E1 17252.288,E2 17252.288} C_VEL
LIN {X 0,Y 376.307,Z 426.917,A -85,B 0,C 180,E1 17250.774,E2 17250.774} C_VEL
LIN {X 0,Y 374.667,Z 410.406,A -85,B 0,C 180,E1 17249.02,E2 17249.02} C_VEL
LIN {X 0,Y 373.797,Z 400.94,A -85,B 0,C 180,E1 17247.837,E2 17247.837} C_VEL
LIN {X 0,Y 380.094,Z 385.902,A -85,B 0,C 180,E1 17244.545,E2 17244.545} C_VEL
LIN {X 0,Y 380.381,Z 381.207,A -85,B 0,C 180,E1 17242.231,E2 17242.231} C_VEL
LIN {X 0,Y 380.652,Z 378.488,A -85,B 0,C 180,E1 17240.086,E2 17240.086} C_VEL
LIN {X 0,Y 381,Z 377.429,A -85,B 0,C 180,E1 17238.186,E2 17238.186} C_VEL
LIN {X 0,Y 381.562,Z 377.458,A -85,B 0,C 180,E1 17236.324,E2 17236.324} C_VEL
LIN {X 0,Y 382.37,Z 379.877,A -85,B 0,C 180,E1 17233.802,E2 17233.802} C_VEL
LIN {X 0,Y 383.085,Z 383.334,A -85,B 0,C 180,E1 17231.927,E2 17231.927} C_VEL
LIN {X 0,Y 383.35,Z 386.066,A -85,B 0,C 180,E1 17230.895,E2 17230.895} C_VEL
LIN {X 0,Y 379.21,Z 396.283,A -85,B 0,C 180,E1 17229.356,E2 17229.356} C_VEL
LIN {X 0,Y 380.078,Z 411.994,A -85,B 0,C 180,E1 17228.152,E2 17228.152} C_VEL
LIN {X 0,Y 380.094,Z 422.655,A -85,B 0,C 180,E1 17227.552,E2 17227.552} C_VEL
LIN {X 0,Y 372.447,Z 501.196,A -85,B 0,C 180,E1 17225.136,E2 17225.136} C_VEL
LIN {X 0,Y 366.395,Z 581.76,A -85,B 0,C 180,E1 17222.777,E2 17222.777} C_VEL
LIN {X 0,Y 364.07,Z 601.397,A -85,B 0,C 180,E1 17221.917,E2 17221.917} C_VEL
LIN {X 0,Y 361.501,Z 618.823,A -85,B 0,C 180,E1 17220.869,E2 17220.869} C_VEL
LIN {X 0,Y 358.613,Z 636.607,A -85,B 0,C 180,E1 17219.48,E2 17219.48} C_VEL
LIN {X 0,Y 355.68,Z 653.498,A -85,B 0,C 180,E1 17217.818,E2 17217.818} C_VEL
LIN {X 0,Y 352.841,Z 669.486,A -85,B 0,C 180,E1 17215.875,E2 17215.875} C_VEL
LIN {X 0,Y 350.215,Z 684.4,A -85,B 0,C 180,E1 17213.65,E2 17213.65} C_VEL
LIN {X 0,Y 348.05,Z 697.797,A -85,B 0,C 180,E1 17211.222,E2 17211.222} C_VEL
LIN {X 0,Y 346.325,Z 710.095,A -85,B 0,C 180,E1 17208.518,E2 17208.518} C_VEL
LIN {X 0,Y 345.252,Z 720.22,A -85,B 0,C 180,E1 17205.798,E2 17205.798} C_VEL
LIN {X 0,Y 344.706,Z 728.917,A -85,B 0,C 180,E1 17202.907,E2 17202.907} C_VEL
LIN {X 0,Y 344.652,Z 736.057,A -85,B 0,C 180,E1 17199.857,E2 17199.857} C_VEL
LIN {X 0,Y 344.906,Z 740.941,A -85,B 0,C 180,E1 17196.995,E2 17196.995} C_VEL
LIN {X 0,Y 345.274,Z 744.102,A -85,B 0,C 180,E1 17194.153,E2 17194.153} C_VEL
LIN {X 0,Y 345.538,Z 745.504,A -85,B 0,C 180,E1 17191.494,E2 17191.494} C_VEL
LIN {X 0,Y 345.59,Z 745.378,A -85,B 0,C 180,E1 17188.841,E2 17188.841} C_VEL
LIN {X 0,Y 345.41,Z 743.692,A -85,B 0,C 180,E1 17186.184,E2 17186.184} C_VEL
LIN {X 0,Y 345.108,Z 740.157,A -85,B 0,C 180,E1 17183.346,E2 17183.346} C_VEL
LIN {X 0,Y 344.867,Z 734.743,A -85,B 0,C 180,E1 17180.489,E2 17180.489} C_VEL
LIN {X 0,Y 344.851,Z 727.625,A -85,B 0,C 180,E1 17177.719,E2 17177.719} C_VEL
LIN {X 0,Y 345.193,Z 718.908,A -85,B 0,C 180,E1 17175.062,E2 17175.062} C_VEL
LIN {X 0,Y 345.91,Z 708.508,A -85,B 0,C 180,E1 17172.507,E2 17172.507} C_VEL
LIN {X 0,Y 347.012,Z 696.656,A -85,B 0,C 180,E1 17170.125,E2 17170.125} C_VEL
LIN {X 0,Y 348.43,Z 683.299,A -85,B 0,C 180,E1 17167.92,E2 17167.92} C_VEL
LIN {X 0,Y 350.126,Z 668.362,A -85,B 0,C 180,E1 17165.899,E2 17165.899} C_VEL
LIN {X 0,Y 351.934,Z 652.464,A -85,B 0,C 180,E1 17164.146,E2 17164.146} C_VEL
LIN {X 0,Y 353.73,Z 635.721,A -85,B 0,C 180,E1 17162.662,E2 17162.662} C_VEL
LIN {X 0,Y 355.427,Z 618.031,A -85,B 0,C 180,E1 17161.432,E2 17161.432} C_VEL
LIN {X 0,Y 356.973,Z 599.31,A -85,B 0,C 180,E1 17160.466,E2 17160.466} C_VEL
LIN {X 0,Y 358.033,Z 580.247,A -85,B 0,C 180,E1 17159.801,E2 17159.801} C_VEL
LIN {X 0,Y 363.287,Z 416.574,A -85,B 0,C 180,E1 17155.94,E2 17155.94} C_VEL
LIN {X 0,Y 360.895,Z 388.87,A -85,B 0,C 180,E1 17155.008,E2 17155.008} C_VEL
LIN {X 0,Y 364.6,Z 362.499,A -85,B 0,C 180,E1 17151.913,E2 17151.913} C_VEL
LIN {X 0,Y 357.162,Z 340.057,A -85,B 0,C 180,E1 17148.222,E2 17148.222} C_VEL
LIN {X 0,Y 350.044,Z 319.588,A -85,B 0,C 180,E1 17144.529,E2 17144.529} C_VEL
LIN {X 0,Y 345.874,Z 307.713,A -85,B 0,C 180,E1 17142.219,E2 17142.219} C_VEL
LIN {X 0,Y 345.885,Z 307.714,A -85,B 0,C 180,E1 17138.007,E2 17138.007} C_VEL
LIN {X 0,Y 345.895,Z 307.714,A -85,B 0,C 180,E1 17133.713,E2 17133.713} C_VEL
LIN {X 0,Y 345.893,Z 307.711,A -85,B 0,C 180,E1 17129.435,E2 17129.435} C_VEL
LIN {X 0,Y 345.879,Z 307.711,A -85,B 0,C 180,E1 17125.206,E2 17125.206} C_VEL
LIN {X 0,Y 345.87,Z 307.711,A -85,B 0,C 180,E1 17120.978,E2 17120.978} C_VEL
LIN {X 0,Y 345.866,Z 307.711,A -85,B 0,C 180,E1 17116.805,E2 17116.805} C_VEL
LIN {X 0,Y 345.865,Z 307.711,A -85,B 0,C 180,E1 17112.524,E2 17112.524} C_VEL
LIN {X 0,Y 345.87,Z 307.711,A -85,B 0,C 180,E1 17108.313,E2 17108.313} C_VEL
LIN {X 0,Y 345.878,Z 307.711,A -85,B 0,C 180,E1 17104.147,E2 17104.147} C_VEL
LIN {X 0,Y 345.883,Z 307.712,A -85,B 0,C 180,E1 17100.002,E2 17100.002} C_VEL
LIN {X 0,Y 345.898,Z 307.712,A -85,B 0,C 180,E1 17095.738,E2 17095.738} C_VEL
LIN {X 0,Y 345.914,Z 307.711,A -85,B 0,C 180,E1 17091.525,E2 17091.525} C_VEL
LIN {X 0,Y 345.903,Z 307.71,A -85,B 0,C 180,E1 17087.312,E2 17087.312} C_VEL
LIN {X 0,Y 345.897,Z 307.71,A -85,B 0,C 180,E1 17083.201,E2 17083.201} C_VEL
LIN {X 0,Y 345.888,Z 307.71,A -85,B 0,C 180,E1 17078.998,E2 17078.998} C_VEL
LIN {X 0,Y 345.884,Z 307.71,A -85,B 0,C 180,E1 17074.857,E2 17074.857} C_VEL
LIN {X 0,Y 345.881,Z 307.709,A -85,B 0,C 180,E1 17070.759,E2 17070.759} C_VEL
LIN {X 0,Y 345.882,Z 307.709,A -85,B 0,C 180,E1 17066.657,E2 17066.657} C_VEL
LIN {X 0,Y 345.879,Z 307.71,A -85,B 0,C 180,E1 17062.377,E2 17062.377} C_VEL
LIN {X 0,Y 345.883,Z 307.709,A -85,B 0,C 180,E1 17058.227,E2 17058.227} C_VEL
LIN {X 0,Y 345.89,Z 307.71,A -85,B 0,C 180,E1 17053.968,E2 17053.968} C_VEL
LIN {X 0,Y 345.901,Z 307.711,A -85,B 0,C 180,E1 17049.75,E2 17049.75} C_VEL
LIN {X 0,Y 345.91,Z 307.712,A -85,B 0,C 180,E1 17045.519,E2 17045.519} C_VEL
LIN {X 0,Y 345.926,Z 307.709,A -85,B 0,C 180,E1 17041.349,E2 17041.349} C_VEL
LIN {X 0,Y 345.917,Z 307.707,A -85,B 0,C 180,E1 17037.102,E2 17037.102} C_VEL
LIN {X 0,Y 345.909,Z 307.707,A -85,B 0,C 180,E1 17032.967,E2 17032.967} C_VEL
LIN {X 0,Y 345.905,Z 307.708,A -85,B 0,C 180,E1 17028.888,E2 17028.888} C_VEL
LIN {X 0,Y 345.898,Z 307.708,A -85,B 0,C 180,E1 17024.735,E2 17024.735} C_VEL
LIN {X 0,Y 345.897,Z 307.708,A -85,B 0,C 180,E1 17020.658,E2 17020.658} C_VEL
LIN {X 0,Y 345.891,Z 307.708,A -85,B 0,C 180,E1 17016.472,E2 17016.472} C_VEL
LIN {X 0,Y 345.889,Z 307.709,A -85,B 0,C 180,E1 17012.152,E2 17012.152} C_VEL
LIN {X 0,Y 345.892,Z 307.709,A -85,B 0,C 180,E1 17008.011,E2 17008.011} C_VEL
LIN {X 0,Y 345.897,Z 307.709,A -85,B 0,C 180,E1 17003.859,E2 17003.859} C_VEL
LIN {X 0,Y 345.904,Z 307.71,A -85,B 0,C 180,E1 16999.675,E2 16999.675} C_VEL
LIN {X 0,Y 345.919,Z 307.711,A -85,B 0,C 180,E1 16995.434,E2 16995.434} C_VEL
LIN {X 0,Y 345.928,Z 307.707,A -85,B 0,C 180,E1 16991.111,E2 16991.111} C_VEL
LIN {X 0,Y 345.925,Z 307.706,A -85,B 0,C 180,E1 16986.852,E2 16986.852} C_VEL
LIN {X 0,Y 345.909,Z 307.706,A -85,B 0,C 180,E1 16982.54,E2 16982.54} C_VEL
LIN {X 0,Y 345.906,Z 307.706,A -85,B 0,C 180,E1 16978.452,E2 16978.452} C_VEL
LIN {X 0,Y 345.901,Z 307.707,A -85,B 0,C 180,E1 16974.273,E2 16974.273} C_VEL
LIN {X 0,Y 345.898,Z 307.708,A -85,B 0,C 180,E1 16969.992,E2 16969.992} C_VEL
LIN {X 0,Y 345.904,Z 307.708,A -85,B 0,C 180,E1 16965.791,E2 16965.791} C_VEL
LIN {X 0,Y 345.913,Z 307.71,A -85,B 0,C 180,E1 16961.526,E2 16961.526} C_VEL
LIN {X 0,Y 345.95,Z 307.802,A -85,B 0,C 180,E1 16960.887,E2 16960.887} C_VEL
LIN {X 0,Y 351.438,Z 327.013,A -85,B 0,C 180,E1 16956.684,E2 16956.684} C_VEL
LIN {X 0,Y 351.684,Z 327.852,A -85,B 0,C 180,E1 16956.507,E2 16956.507} C_VEL
LIN {X 0,Y 352.053,Z 332.894,A -85,B 0,C 180,E1 16955.549,E2 16955.549} C_VEL
LIN {X 0,Y 349.419,Z 348.469,A -85,B 0,C 180,E1 16952.946,E2 16952.946} C_VEL
LIN {X 0,Y 349.757,Z 352.134,A -85,B 0,C 180,E1 16952.257,E2 16952.257} C_VEL
LIN {X 0,Y 347.732,Z 369.917,A -85,B 0,C 180,E1 16949.259,E2 16949.259} C_VEL
LIN {X 0,Y 344.575,Z 398.091,A -85,B 0,C 180,E1 16944.577,E2 16944.577} C_VEL
LIN {X 0,Y 344.227,Z 402.038,A -85,B 0,C 180,E1 16943.983,E2 16943.983} C_VEL
LIN {X 0,Y 348.082,Z 435.565,A -85,B 0,C 180,E1 16942.672,E2 16942.672} C_VEL
LIN {X 0,Y 344.251,Z 532.161,A -85,B 0,C 180,E1 16939.757,E2 16939.757} C_VEL
LIN {X 0,Y 343.549,Z 548.639,A -85,B 0,C 180,E1 16938.966,E2 16938.966} C_VEL
LIN {X 0,Y 342.647,Z 565.287,A -85,B 0,C 180,E1 16937.839,E2 16937.839} C_VEL
LIN {X 0,Y 341.606,Z 581.223,A -85,B 0,C 180,E1 16936.404,E2 16936.404} C_VEL
LIN {X 0,Y 340.596,Z 595.803,A -85,B 0,C 180,E1 16934.707,E2 16934.707} C_VEL
LIN {X 0,Y 339.64,Z 609.03,A -85,B 0,C 180,E1 16932.753,E2 16932.753} C_VEL
LIN {X 0,Y 338.881,Z 619.993,A -85,B 0,C 180,E1 16930.71,E2 16930.71} C_VEL
LIN {X 0,Y 338.356,Z 628.805,A -85,B 0,C 180,E1 16928.665,E2 16928.665} C_VEL
LIN {X 0,Y 337.995,Z 636.753,A -85,B 0,C 180,E1 16926.281,E2 16926.281} C_VEL
LIN {X 0,Y 337.86,Z 642.621,A -85,B 0,C 180,E1 16923.9,E2 16923.9} C_VEL
LIN {X 0,Y 337.944,Z 646.7,A -85,B 0,C 180,E1 16921.523,E2 16921.523} C_VEL
LIN {X 0,Y 338.243,Z 649.116,A -85,B 0,C 180,E1 16918.981,E2 16918.981} C_VEL
LIN {X 0,Y 338.753,Z 649.693,A -85,B 0,C 180,E1 16916.613,E2 16916.613} C_VEL
LIN {X 0,Y 339.506,Z 648.556,A -85,B 0,C 180,E1 16914.251,E2 16914.251} C_VEL
LIN {X 0,Y 340.623,Z 645.484,A -85,B 0,C 180,E1 16911.728,E2 16911.728} C_VEL
LIN {X 0,Y 342.004,Z 640.766,A -85,B 0,C 180,E1 16909.384,E2 16909.384} C_VEL
LIN {X 0,Y 343.747,Z 634.126,A -85,B 0,C 180,E1 16907.056,E2 16907.056} C_VEL
LIN {X 0,Y 345.868,Z 625.233,A -85,B 0,C 180,E1 16904.746,E2 16904.746} C_VEL
LIN {X 0,Y 348,Z 615.516,A -85,B 0,C 180,E1 16902.784,E2 16902.784} C_VEL
LIN {X 0,Y 350.439,Z 603.452,A -85,B 0,C 180,E1 16900.844,E2 16900.844} C_VEL
LIN {X 0,Y 352.977,Z 589.512,A -85,B 0,C 180,E1 16899.087,E2 16899.087} C_VEL
LIN {X 0,Y 355.57,Z 573.669,A -85,B 0,C 180,E1 16897.514,E2 16897.514} C_VEL
LIN {X 0,Y 357.851,Z 557.326,A -85,B 0,C 180,E1 16896.273,E2 16896.273} C_VEL
LIN {X 0,Y 359.935,Z 539.894,A -85,B 0,C 180,E1 16895.277,E2 16895.277} C_VEL
LIN {X 0,Y 368.396,Z 475.321,A -85,B 0,C 180,E1 16892.559,E2 16892.559} C_VEL
LIN {X 0,Y 372.572,Z 446.336,A -85,B 0,C 180,E1 16891.364,E2 16891.364} C_VEL
LIN {X 0,Y 371.748,Z 429.536,A -85,B 0,C 180,E1 16889.825,E2 16889.825} C_VEL
LIN {X 0,Y 370.577,Z 414.28,A -85,B 0,C 180,E1 16888.129,E2 16888.129} C_VEL
LIN {X 0,Y 369.712,Z 400.684,A -85,B 0,C 180,E1 16886.328,E2 16886.328} C_VEL
LIN {X 0,Y 374.384,Z 390.565,A -85,B 0,C 180,E1 16884.015,E2 16884.015} C_VEL
LIN {X 0,Y 374.865,Z 386.389,A -85,B 0,C 180,E1 16881.77,E2 16881.77} C_VEL
LIN {X 0,Y 375.396,Z 383.802,A -85,B 0,C 180,E1 16879.386,E2 16879.386} C_VEL
LIN {X 0,Y 376.134,Z 383.252,A -85,B 0,C 180,E1 16876.697,E2 16876.697} C_VEL
LIN {X 0,Y 376.899,Z 385.517,A -85,B 0,C 180,E1 16874.032,E2 16874.032} C_VEL
LIN {X 0,Y 377.568,Z 389.101,A -85,B 0,C 180,E1 16872.067,E2 16872.067} C_VEL
LIN {X 0,Y 377.568,Z 390.75,A -85,B 0,C 180,E1 16871.457,E2 16871.457} C_VEL
LIN {X 0,Y 375.012,Z 396.805,A -85,B 0,C 180,E1 16870.532,E2 16870.532} C_VEL
LIN {X 0,Y 375.588,Z 412.56,A -85,B 0,C 180,E1 16869.223,E2 16869.223} C_VEL
LIN {X 0,Y 375.49,Z 423.726,A -85,B 0,C 180,E1 16868.532,E2 16868.532} C_VEL
LIN {X 0,Y 367.144,Z 500.904,A -85,B 0,C 180,E1 16866.076,E2 16866.076} C_VEL
LIN {X 0,Y 360.437,Z 580.616,A -85,B 0,C 180,E1 16863.645,E2 16863.645} C_VEL
LIN {X 0,Y 358.032,Z 599.551,A -85,B 0,C 180,E1 16862.806,E2 16862.806} C_VEL
LIN {X 0,Y 355.104,Z 617.992,A -85,B 0,C 180,E1 16861.678,E2 16861.678} C_VEL
LIN {X 0,Y 351.847,Z 636.409,A -85,B 0,C 180,E1 16860.199,E2 16860.199} C_VEL
LIN {X 0,Y 348.588,Z 653.736,A -85,B 0,C 180,E1 16858.435,E2 16858.435} C_VEL
LIN {X 0,Y 345.44,Z 669.88,A -85,B 0,C 180,E1 16856.38,E2 16856.38} C_VEL
LIN {X 0,Y 342.653,Z 684.451,A -85,B 0,C 180,E1 16854.113,E2 16854.113} C_VEL
LIN {X 0,Y 340.273,Z 698.006,A -85,B 0,C 180,E1 16851.55,E2 16851.55} C_VEL
LIN {X 0,Y 338.448,Z 710.031,A -85,B 0,C 180,E1 16848.786,E2 16848.786} C_VEL
LIN {X 0,Y 337.253,Z 720.477,A -85,B 0,C 180,E1 16845.829,E2 16845.829} C_VEL
LIN {X 0,Y 336.705,Z 728.817,A -85,B 0,C 180,E1 16842.87,E2 16842.87} C_VEL
LIN {X 0,Y 336.668,Z 735.301,A -85,B 0,C 180,E1 16839.92,E2 16839.92} C_VEL
LIN {X 0,Y 336.951,Z 740.031,A -85,B 0,C 180,E1 16836.989,E2 16836.989} C_VEL
LIN {X 0,Y 337.354,Z 743.048,A -85,B 0,C 180,E1 16834.08,E2 16834.08} C_VEL
LIN {X 0,Y 337.636,Z 744.338,A -85,B 0,C 180,E1 16831.359,E2 16831.359} C_VEL
LIN {X 0,Y 337.682,Z 744.032,A -85,B 0,C 180,E1 16828.644,E2 16828.644} C_VEL
LIN {X 0,Y 337.486,Z 742.151,A -85,B 0,C 180,E1 16825.924,E2 16825.924} C_VEL
LIN {X 0,Y 337.175,Z 738.66,A -85,B 0,C 180,E1 16823.189,E2 16823.189} C_VEL
LIN {X 0,Y 336.931,Z 733.484,A -85,B 0,C 180,E1 16820.435,E2 16820.435} C_VEL
LIN {X 0,Y 336.904,Z 726.506,A -85,B 0,C 180,E1 16817.663,E2 16817.663} C_VEL
LIN {X 0,Y 337.225,Z 718.156,A -85,B 0,C 180,E1 16815.053,E2 16815.053} C_VEL
LIN {X 0,Y 337.943,Z 707.811,A -85,B 0,C 180,E1 16812.437,E2 16812.437} C_VEL
LIN {X 0,Y 339.061,Z 696.024,A -85,B 0,C 180,E1 16809.998,E2 16809.998} C_VEL
LIN {X 0,Y 340.507,Z 682.764,A -85,B 0,C 180,E1 16807.743,E2 16807.743} C_VEL
